   STATUS[3878] := 16#00;
   STATUS[3879] := 16#00;
   STATUS[3880] := 16#00;
   STATUS[3881] := 16#00;
   STATUS[3882] := 16#00;
   STATUS[3883] := 16#00;
   STATUS[3884] := 16#00;
   STATUS[3885] := 16#00;
   STATUS[3886] := 16#00;
   STATUS[3887] := 16#00;
   STATUS[3888] := 16#00;
   STATUS[3889] := 16#00;
   STATUS[3890] := 16#00;
   STATUS[3891] := 16#00;
   STATUS[3892] := 16#00;
   STATUS[3893] := 16#00;
   STATUS[3894] := 16#00;
   STATUS[3895] := 16#00;
   STATUS[3896] := 16#00;
   STATUS[3897] := 16#00;
   STATUS[3898] := 16#00;
   STATUS[3899] := 16#00;
   STATUS[3900] := 16#00;
   STATUS[3901] := 16#00;
   STATUS[3902] := 16#00;
   STATUS[3903] := 16#00;
   STATUS[3904] := 16#00;
   STATUS[3905] := 16#00;
   STATUS[3906] := 16#00;
   STATUS[3907] := 16#00;
   STATUS[3908] := 16#00;
   STATUS[3909] := 16#00;
   STATUS[3910] := 16#00;
   STATUS[3911] := 16#00;
   STATUS[3912] := 16#00;
   STATUS[3913] := 16#00;
   STATUS[3914] := 16#00;
   STATUS[3915] := 16#00;
   STATUS[3916] := 16#00;
   STATUS[3917] := 16#00;
   STATUS[3918] := 16#00;
   STATUS[3919] := 16#00;
   STATUS[3920] := 16#00;
   STATUS[3921] := 16#00;
   STATUS[3922] := 16#00;
   STATUS[3923] := 16#00;
   STATUS[3924] := 16#00;
   STATUS[3925] := 16#00;
   STATUS[3926] := 16#00;
   STATUS[3927] := 16#00;
   STATUS[3928] := 16#00;
   STATUS[3929] := 16#00;
   STATUS[3930] := 16#00;
   STATUS[3931] := 16#00;
   STATUS[3932] := 16#00;
   STATUS[3933] := 16#00;
   STATUS[3934] := 16#00;
   STATUS[3935] := 16#00;
   STATUS[3936] := 16#00;
   STATUS[3937] := 16#00;
   STATUS[3938] := 16#00;
   STATUS[3939] := 16#00;
   STATUS[3940] := 16#00;
   STATUS[3941] := 16#00;
   STATUS[3942] := 16#00;
   STATUS[3943] := 16#00;
   STATUS[3944] := 16#00;
   STATUS[3945] := 16#00;
   STATUS[3946] := 16#00;
   STATUS[3947] := 16#00;
   STATUS[3948] := 16#00;
   STATUS[3949] := 16#00;
   STATUS[3950] := 16#00;
   STATUS[3951] := 16#00;
   STATUS[3952] := 16#00;
   STATUS[3953] := 16#00;
   STATUS[3954] := 16#00;
   STATUS[3955] := 16#00;
   STATUS[3956] := 16#00;
   STATUS[3957] := 16#00;
   STATUS[3958] := 16#00;
   STATUS[3959] := 16#00;
   STATUS[3960] := 16#00;
   STATUS[3961] := 16#00;
   STATUS[3962] := 16#00;
   STATUS[3963] := 16#00;
   STATUS[3964] := 16#00;
   STATUS[3965] := 16#00;
   STATUS[3966] := 16#00;
   STATUS[3967] := 16#00;
   STATUS[3968] := 16#00;
   STATUS[3969] := 16#00;
   STATUS[3970] := 16#00;
   STATUS[3971] := 16#00;
   STATUS[3972] := 16#00;
   STATUS[3973] := 16#00;
   STATUS[3974] := 16#00;
   STATUS[3975] := 16#00;
   STATUS[3976] := 16#00;
   STATUS[3977] := 16#00;
   STATUS[3978] := 16#00;
   STATUS[3979] := 16#00;
   STATUS[3980] := 16#00;
   STATUS[3981] := 16#00;
   STATUS[3982] := 16#00;
   STATUS[3983] := 16#00;
   STATUS[3984] := 16#00;
   STATUS[3985] := 16#00;
   STATUS[3986] := 16#00;
   STATUS[3987] := 16#00;
   STATUS[3988] := 16#00;
   STATUS[3989] := 16#00;
   STATUS[3990] := 16#00;
   STATUS[3991] := 16#00;
   STATUS[3992] := 16#00;
   STATUS[3993] := 16#00;
   STATUS[3994] := 16#00;
   STATUS[3995] := 16#00;
   STATUS[3996] := 16#00;
   STATUS[3997] := 16#00;
   STATUS[3998] := 16#00;
   STATUS[3999] := 16#00;
   STATUS[4000] := 16#00;
   STATUS[4001] := 16#00;
   STATUS[4002] := 16#00;
   STATUS[4003] := 16#00;
   STATUS[4004] := 16#00;
   STATUS[4005] := 16#00;
   STATUS[4006] := 16#00;
   STATUS[4007] := 16#00;
   STATUS[4008] := 16#00;
   STATUS[4009] := 16#00;
   STATUS[4010] := 16#00;
   STATUS[4011] := 16#00;
   STATUS[4012] := 16#00;
   STATUS[4013] := 16#00;
   STATUS[4014] := 16#00;
   STATUS[4015] := 16#00;
   STATUS[4016] := 16#00;
   STATUS[4017] := 16#00;
   STATUS[4018] := 16#00;
   STATUS[4019] := 16#00;
   STATUS[4020] := 16#00;
   STATUS[4021] := 16#00;
   STATUS[4022] := 16#00;
   STATUS[4023] := 16#00;
   STATUS[4024] := 16#00;
   STATUS[4025] := 16#00;
   STATUS[4026] := 16#00;
   STATUS[4027] := 16#00;
   STATUS[4028] := 16#00;
   STATUS[4029] := 16#00;
   STATUS[4030] := 16#00;
   STATUS[4031] := 16#00;
   STATUS[4032] := 16#00;
   STATUS[4033] := 16#00;
   STATUS[4034] := 16#00;
   STATUS[4035] := 16#00;
   STATUS[4036] := 16#00;
   STATUS[4037] := 16#00;
   STATUS[4038] := 16#00;
   STATUS[4039] := 16#00;
   STATUS[4040] := 16#00;
   STATUS[4041] := 16#00;
   STATUS[4042] := 16#00;
   STATUS[4043] := 16#00;
   STATUS[4044] := 16#00;
   STATUS[4045] := 16#00;
   STATUS[4046] := 16#00;
   STATUS[4047] := 16#00;
   STATUS[4048] := 16#00;
   STATUS[4049] := 16#00;
   STATUS[4050] := 16#00;
   STATUS[4051] := 16#00;
   STATUS[4052] := 16#00;
   STATUS[4053] := 16#00;
   STATUS[4054] := 16#00;
   STATUS[4055] := 16#00;
   STATUS[4056] := 16#00;
   STATUS[4057] := 16#00;
   STATUS[4058] := 16#00;
   STATUS[4059] := 16#00;
   STATUS[4060] := 16#00;
   STATUS[4061] := 16#00;
   STATUS[4062] := 16#00;
   STATUS[4063] := 16#00;
   STATUS[4064] := 16#00;
   STATUS[4065] := 16#00;
   STATUS[4066] := 16#00;
   STATUS[4067] := 16#00;
   STATUS[4068] := 16#00;
   STATUS[4069] := 16#00;
   STATUS[4070] := 16#00;
   STATUS[4071] := 16#00;
   STATUS[4072] := 16#00;
   STATUS[4073] := 16#00;
   STATUS[4074] := 16#00;
   STATUS[4075] := 16#00;
   STATUS[4076] := 16#00;
   STATUS[4077] := 16#00;
   STATUS[4078] := 16#00;
   STATUS[4079] := 16#00;
   STATUS[4080] := 16#00;
   STATUS[4081] := 16#00;
   STATUS[4082] := 16#00;
   STATUS[4083] := 16#00;
   STATUS[4084] := 16#00;
   STATUS[4085] := 16#00;
   STATUS[4086] := 16#00;
   STATUS[4087] := 16#00;
   STATUS[4088] := 16#00;
   STATUS[4089] := 16#00;
   STATUS[4090] := 16#00;
   STATUS[4091] := 16#00;
   STATUS[4092] := 16#00;
   STATUS[4093] := 16#00;
   STATUS[4094] := 16#00;
   STATUS[4095] := 16#00;
   STATUS[4096] := 16#00;
END_DATA_BLOCK

DATA_BLOCK "ACESYS_HMI_INDICATION"   // DB11
TITLE = Boolean Indications to HMI
{ S7_Optimized_Access := 'FALSE' }
AUTHOR : METIS
FAMILY : ACESYS
NAME : IndDB
VERSION : 8.0
   VAR
      "997CD100D01_RESET_ALRM" : Bool := FALSE;   // Reset Alarm In Area
      "2010BF110U01_STOP_FROM_ECS" : Bool := FALSE;   // Ext Stop From ECS
      "2010HP100TL01CMD01" : Bool := FALSE;   // Переключение сигнала сфетофора
      "2010HP100TL01GRN01" : Bool := FALSE;   // Светофор красный
      "2010HP100TL01RED01" : Bool := TRUE;   // Светофор красный
      "2010BF110U01_SPD_UP" : Bool := FALSE;   // Увеличить задание на 1
      "2010BF110U01_SPD_DN" : Bool := TRUE;   // Уменьшить задание на 1
      "3015PU040_042_OFF" : Bool := FALSE;
      "2010HP100TL01CMD2" : Bool := FALSE;   // Светофор Включить зелёный
      "2010HP100TL01CMD3" : Bool := FALSE;   // Светофор Включить красный
      IND11 : Bool := FALSE;
      IND12 : Bool := TRUE;
      IND13 : Bool := FALSE;
      IND14 : Bool := FALSE;
      IND15 : Bool := FALSE;
      IND16 : Bool := TRUE;
      IND17 : Bool := FALSE;
      IND18 : Bool := FALSE;
      IND19 : Bool := FALSE;
      "2010SJ950M01_ASTR" : Bool := FALSE;
      IND21 : Bool := FALSE;
      IND22 : Bool := FALSE;
      IND23 : Bool := FALSE;
      IND24 : Bool := FALSE;
      IND25 : Bool := FALSE;
      IND26 : Bool := FALSE;
      IND27 : Bool := FALSE;
      IND28 : Bool := TRUE;
      IND29 : Bool := FALSE;
      IND30 : Bool := FALSE;
      IND31 : Bool := FALSE;
      IND32 : Bool := FALSE;
      IND33 : Bool := FALSE;
      IND34 : Bool := FALSE;
      IND35 : Bool := FALSE;
      IND36 : Bool := FALSE;
      IND37 : Bool := FALSE;
      IND38 : Bool := FALSE;
      IND39 : Bool := FALSE;
      IND40 : Bool := FALSE;
      IND41 : Bool := FALSE;
      IND42 : Bool := FALSE;
      IND43 : Bool := TRUE;
      IND44 : Bool := TRUE;
      IND45 : Bool := FALSE;
      IND46 : Bool := FALSE;
      IND47 : Bool := FALSE;
      IND48 : Bool := FALSE;
      IND49 : Bool := FALSE;
      IND50 : Bool := FALSE;
      IND51 : Bool := FALSE;
      IND52 : Bool := FALSE;
      IND53 : Bool := FALSE;
      IND54 : Bool := TRUE;
      IND55 : Bool := FALSE;
      IND56 : Bool := TRUE;
      IND57 : Bool := TRUE;
      IND58 : Bool := TRUE;
      IND59 : Bool := FALSE;
      _995CS100_INDICATION01 : Bool := FALSE;   // INDICATION01
      _995CS100_INDICATION02 : Bool := FALSE;   // INDICATION02
      _995CS100_INDICATION03 : Bool := FALSE;   // INDICATION03
      _995CS100_INDICATION04 : Bool := FALSE;   // INDICATION04
      _995CS100_INDICATION05 : Bool := FALSE;   // INDICATION05
      _995CS100_INDICATION06 : Bool := FALSE;   // INDICATION06
      _995CS100_INDICATION07 : Bool := FALSE;   // INDICATION07
      _995CS100_INDICATION08 : Bool := FALSE;   // INDICATION08
      _995CS100_INDICATION09 : Bool := FALSE;   // INDICATION09
      _995CS100_INDICATION10 : Bool := FALSE;   // INDICATION10
      _995CS100_INDICATION11 : Bool := FALSE;   // INDICATION11
      _995CS100_INDICATION12 : Bool := FALSE;   // INDICATION12
      _995CS100_INDICATION13 : Bool := FALSE;   // INDICATION13
      _995CS100_INDICATION14 : Bool := FALSE;   // INDICATION14
      _995CS100_INDICATION15 : Bool := FALSE;   // INDICATION15
      _995CS100_INDICATION16 : Bool := FALSE;   // INDICATION16
      _995CS100_INDICATION17 : Bool := FALSE;   // INDICATION17
      _995CS100_INDICATION18 : Bool := FALSE;   // INDICATION18
      _995CS100_INDICATION19 : Bool := FALSE;   // INDICATION19
      _995CS100_INDICATION20 : Bool := FALSE;   // INDICATION20
      _995CS100_INDICATION21 : Bool := FALSE;   // INDICATION21
      _995CS100_INDICATION22 : Bool := FALSE;   // INDICATION22
      _995CS100_INDICATION23 : Bool := FALSE;   // INDICATION23
      _995CS100_INDICATION24 : Bool := FALSE;   // INDICATION24
      _995CS100_INDICATION25 : Bool := FALSE;   // INDICATION25
      _995CS100_INDICATION26 : Bool := FALSE;   // INDICATION26
      _995CS100_INDICATION27 : Bool := FALSE;   // INDICATION27
      _995CS100_INDICATION28 : Bool := FALSE;   // INDICATION28
      _995CS100_INDICATION29 : Bool := FALSE;   // INDICATION29
      _995CS100_INDICATION30 : Bool := FALSE;   // INDICATION30
      _995CS100_INDICATION31 : Bool := FALSE;   // INDICATION31
      _995CS100_INDICATION32 : Bool := FALSE;   // INDICATION32
      _995CS100_INDICATION33 : Bool := FALSE;   // INDICATION33
      _995CS100_INDICATION34 : Bool := FALSE;   // INDICATION34
      _995CS100_INDICATION35 : Bool := FALSE;   // INDICATION35
      _995CS100_INDICATION36 : Bool := FALSE;   // INDICATION36
      _995CS100_INDICATION37 : Bool := FALSE;   // INDICATION37
      _995CS100_INDICATION38 : Bool := FALSE;   // INDICATION38
      _995CS100_INDICATION39 : Bool := FALSE;   // INDICATION39
      _995CS100_INDICATION40 : Bool := FALSE;   // INDICATION40
      _995CS100_INDICATION41 : Bool := FALSE;   // INDICATION41
      _995CS100_INDICATION42 : Bool := FALSE;   // INDICATION42
      _995CS100_INDICATION43 : Bool := FALSE;   // INDICATION43
      _995CS100_INDICATION44 : Bool := FALSE;   // INDICATION44
      _995CS100_INDICATION45 : Bool := FALSE;   // INDICATION45
      _995CS100_INDICATION46 : Bool := FALSE;   // INDICATION46
      _995CS100_INDICATION47 : Bool := FALSE;   // INDICATION47
      _995CS100_INDICATION48 : Bool := FALSE;   // INDICATION48
      _995CS100_INDICATION49 : Bool := FALSE;   // INDICATION49
      _995CS100_INDICATION50 : Bool := FALSE;   // INDICATION50
      _995CS100_SIMPLEINDI01 : Bool := FALSE;   // SIMPLEINDI01
      _995CS100_SIMPLEINDI02 : Bool := FALSE;   // SIMPLEINDI02
      _995CS100_SIMPLEINDI03 : Bool := FALSE;   // SIMPLEINDI03
      _995CS100_SIMPLEINDI04 : Bool := FALSE;   // SIMPLEINDI04
      _995CS100_SIMPLEINDI05 : Bool := FALSE;   // SIMPLEINDI05
      _995CS100_SIMPLEINDI06 : Bool := FALSE;   // SIMPLEINDI06
      _995CS100_SIMPLEINDI07 : Bool := FALSE;   // SIMPLEINDI07
      _995CS100_SIMPLEINDI08 : Bool := FALSE;   // SIMPLEINDI08
      _995CS100_SIMPLEINDI09 : Bool := FALSE;   // SIMPLEINDI09
      _995CS100_SIMPLEINDI10 : Bool := FALSE;   // SIMPLEINDI10
      _995CS100_SIMPLEINDI11 : Bool := FALSE;   // SIMPLEINDI11
      _995CS100_SIMPLEINDI12 : Bool := FALSE;   // SIMPLEINDI12
      _995CS100_SIMPLEINDI13 : Bool := FALSE;   // SIMPLEINDI13
      _995CS100_SIMPLEINDI14 : Bool := FALSE;   // SIMPLEINDI14
      _995CS100_SIMPLEINDI15 : Bool := FALSE;   // SIMPLEINDI15
      _995CS100_SIMPLEINDI16 : Bool := FALSE;   // SIMPLEINDI16
      _995CS100_SIMPLEINDI17 : Bool := FALSE;   // SIMPLEINDI17
      _995CS100_SIMPLEINDI18 : Bool := FALSE;   // SIMPLEINDI18
      _995CS100_SIMPLEINDI19 : Bool := FALSE;   // SIMPLEINDI19
      _995CS100_SIMPLEINDI20 : Bool := FALSE;   // SIMPLEINDI20
   END_VAR
BEGIN
END_DATA_BLOCK

DATA_BLOCK "ACESYS_HMI_OPERATORSP"   // DB12
TITLE = Simple setpoints from HMI
{ S7_Optimized_Access := 'FALSE' }
AUTHOR : METIS
FAMILY : ACESYS
NAME : OpDB
VERSION : 8.0
   VAR
      _2010CV300U01_SP : Real := 120.0;   // Set Spd CV300
      _2010CV180U01_SP : Real := 100.0;   // Set Speed
      _spare : Real := 0.0;   // Set Speed
      _2010BF110U01_SP : Real := 0.0;   // Set Speed
      _2010SC130U01_SP : Real := 100.0;   // Set Speed
      _MTR_SPARE_SP : Real := 110.0;
      spare_6 : Real := 70.0;
      spare_7 : Real := 0.0;
      spare_8 : Real := 0.0;
      spare_9 : Real := 0.0;
      spare_10 : Real := 0.0;
      spare_11 : Real := 0.0;
      spare_12 : Real := 0.0;
      spare_13 : Real := 0.0;
      spare_14 : Real := 0.0;   // OPERATORSP01
      spare_15 : Real := 0.0;   // OPERATORSP02
      spare_16 : Real := 0.0;   // OPERATORSP03
      spare_17 : Real := 0.0;   // OPERATORSP04
      spare_18 : Real := 0.0;   // OPERATORSP05
      spare_19 : Real := 0.0;   // OPERATORSP06
      spare_20 : Real := 0.0;   // OPERATORSP07
      spare_21 : Real := 0.0;   // OPERATORSP08
      spare_22 : Real := 0.0;   // OPERATORSP09
      spare_23 : Real := 0.0;   // OPERATORSP10
      spare_24 : Real := 0.0;   // OPERATORSP11
      spare_25 : Real := 0.0;   // OPERATORSP12
      spare_26 : Real := 0.0;   // OPERATORSP13
      spare_27 : Real := 0.0;   // OPERATORSP14
      spare_28 : Real := 0.0;   // OPERATORSP15
      spare_29 : Real := 0.0;   // OPERATORSP16
      spare_30 : Real := 0.0;   // OPERATORSP17
      spare_31 : Real := 0.0;   // OPERATORSP18
      spare_32 : Real := 0.0;   // OPERATORSP19
      spare_33 : Real := 0.0;   // OPERATORSP20
      spare_34 : Real := 0.0;   // OPERATORSP21
      spare_35 : Real := 0.0;   // OPERATORSP22
      spare_36 : Real := 0.0;   // OPERATORSP23
      spare_37 : Real := 0.0;   // OPERATORSP24
      spare_38 : Real := 0.0;   // OPERATORSP25
      spare_39 : Real := 0.0;   // OPERATORSP26
      spare_40 : Real := 0.0;   // OPERATORSP27
      spare_41 : Real := 0.0;   // OPERATORSP28
      spare_42 : Real := 0.0;   // OPERATORSP29
      spare_43 : Real := 0.0;   // OPERATORSP30
   END_VAR
BEGIN
END_DATA_BLOCK

DATA_BLOCK "ACESYS_HMI_SIMPLEAI"   // DB13
TITLE = Simple Analog Values to HMI
{ S7_Optimized_Access := 'FALSE' }
AUTHOR : METIS
FAMILY : ACESYS
NAME : AiDB
VERSION : 8.0
   VAR
      _997CS100_Sec : Real := 16#0000_001A;   // CPU Clock Seconds
      _997CS100_Min : Real := 16#0000_0009;   // CPU Clock Minutes
      _997CS100_Hour : Real := 16#0000_000E;   // CPU Clock Hours
      _997CS100_Day : Real := 16#0000_0009;   // CPU Clock Day
      _997CS100_Month : Real := 16#0000_0003;   // CPU Clock Month
      _997CS100_Year : Real := 16#0000_0019;   // CPU Clock Year
      _997CS100_MemTot : Real := 1.884792E-29;   // Total CPU Memory
      _997CS100_MemUsed : Real := 1.715889E-38;   // Used CPU Memory
      _997CS100_MemPct : Real := 4.63501;   // Used CPU Memory
      _2015PU040U01_AO1b : Real := 10.64;
      _2015PU040U01_AO3a : Real := 80.005;
      _2015PU041U01_AO1b : Real := 0.0;
      _2015PU041U01_AO3a : Real := 0.0;
      _2015PU042U01_AO1b : Real := 4.361;
      _2015PU027U01_AO1b : Real := 0.0;
      _2015PU027U01_AO3a : Real := 0.0;
      _2015PU028U01_AO1b : Real := 0.0;
      _2015PU028U01_AO3a : Real := 0.0;
      _2015PU035U01_AO1b : Real := 0.0;
      _2015PU035U01_AO3a : Real := 0.0;
      _2010SJ950M01_AO1b : Real := 0.0;
      _993CS100_ANALOGINDI22 : Real := 700.0326;
      _993CS100_ANALOGINDI23 : Real := 0.0;
      _993CS100_ANALOGINDI24 : Real := 0.0;
      _993CS100_ANALOGINDI25 : Real := 0.0;
      _993CS100_ANALOGINDI26 : Real := 0.0;
      _993CS100_ANALOGINDI27 : Real := 0.0;
      _993CS100_ANALOGINDI28 : Real := 0.0;
      _993CS100_ANALOGINDI29 : Real := 0.0;
      _993CS100_ANALOGINDI30 : Real := 0.0;
      _993CS100_ANALOGINDI31 : Real := 0.0;
      _993CS100_ANALOGINDI32 : Real := 0.0;
      _993CS100_ANALOGINDI33 : Real := 0.0;
      _993CS100_ANALOGINDI34 : Real := 0.0;
      _993CS100_ANALOGINDI35 : Real := 0.0;
      _993CS100_ANALOGINDI36 : Real := 0.0;
      _993CS100_ANALOGINDI37 : Real := 0.0;
      _993CS100_ANALOGINDI38 : Real := 0.0;
      _993CS100_ANALOGINDI39 : Real := 0.0;
      _993CS100_ANALOGINDI40 : Real := 0.0;
      _993CS100_ANALOGINDI41 : Real := 0.0;
      _993CS100_ANALOGINDI42 : Real := 0.0;
      _993CS100_ANALOGINDI43 : Real := 0.0;
      _993CS100_ANALOGINDI44 : Real := 0.0;
      _993CS100_ANALOGINDI45 : Real := 0.0;
      _993CS100_ANALOGINDI46 : Real := 0.0;
      _993CS100_ANALOGINDI47 : Real := 0.0;
      _993CS100_ANALOGINDI48 : Real := 0.0;
      _993CS100_ANALOGINDI49 : Real := 0.0;
      _993CS100_ANALOGINDI50 : Real := 16#0000_003C;   // OB1 Scan Time
      _993CS100_ANALOGINDI51 : Real := 16#0000_0064;   // OB35 Scan Time
      _993CS100_ANALOGINDI52 : Real := 0.0;
      _993CS100_ANALOGINDI53 : Real := 0.0;
      _993CS100_ANALOGINDI54 : Real := 0.0;
      _993CS100_ANALOGINDI55 : Real := 0.0;
      _993CS100_ANALOGINDI56 : Real := 0.0;
      _993CS100_ANALOGINDI57 : Real := 0.0;
      _993CS100_ANALOGINDI58 : Real := 0.0;
      _993CS100_ANALOGINDI59 : Real := 0.0;
      _2010LV100P01_I1 : Real := 7.9433;
      _2010LV100P01_I2 : Real := 9.236307;
      _2010LV100P01_I3 : Real := 6.303556;
      _2010LV100P01_E01 : Real := 412.6258;
      _2010LV100P01_E02 : Real := 411.3553;
      _2010LV100P01_E03 : Real := 412.2155;
      _2010LV100P01_X01 : Real := 49.99622;
      _2010LV100P01_X02 : Real := 0.8079877;
      _2010LV100P01_J1 : Real := 5.585882;
      _2010LV100P01_J2 : Real := 4.513324;
      _2010LV100P01_J3 : Real := 2.662353;
      _2010LV100P01_Q01 : Real := 1852637.0;
      _2010LV100P01_Q02 : Real := 355350.2;
      _2010LV100P01_Q03 : Real := 2301733.0;
      _993CS100_ANALOGINDI74 : Real := 0.0;
      _993CS100_ANALOGINDI75 : Real := 0.0;
      _993CS100_ANALOGINDI76 : Real := 0.0;
      _993CS100_ANALOGINDI77 : Real := 0.0;
      _993CS100_ANALOGINDI78 : Real := 0.0;
      _993CS100_ANALOGINDI79 : Real := 0.0;
      _993CS100_ANALOGINDI80 : Real := 0.0;
      _993CS100_ANALOGINDI81 : Real := 0.0;
   END_VAR
BEGIN
END_DATA_BLOCK

DATA_BLOCK "ACESYS_HMI_SIMPLEREQ"   // DB14
TITLE = Simple Binary Requests from HMI
{ S7_Optimized_Access := 'FALSE' }
AUTHOR : METIS
FAMILY : ACESYS
NAME : BinReq
VERSION : 8.0
   VAR
      _995CS100HLC_CCA1 : Bool := FALSE;   // Computer Control Accept (Group 1-5)
      _995CS100HLC_CCA1_1 : Bool := FALSE;   // Dont use Bit 1
      _995CS100HLC_CCA1_2 : Bool := FALSE;   // Dont use Bit 2
      _995CS100HLC_CCA1_3 : Bool := FALSE;   // Dont use Bit 3
      _995CS100HLC_CCA1_4 : Bool := FALSE;   // Dont use Bit 4
      _995CS100HLC_CCA1_5 : Bool := FALSE;   // Dont use Bit 5
      _995CS100HLC_CCA1_6 : Bool := FALSE;   // Dont use Bit 6
      _995CS100HLC_CCA1_7 : Bool := FALSE;   // Dont use Bit 7
      _995CS100HLC_CCA2 : Bool := FALSE;   // Computer Control Accept (Group 6-10)
      _995CS100HLC_CCA2_1 : Bool := FALSE;   // Dont use Bit 1
      _995CS100HLC_CCA2_2 : Bool := FALSE;   // Dont use Bit 2
      _995CS100HLC_CCA2_3 : Bool := FALSE;   // Dont use Bit 3
      _995CS100HLC_CCA2_4 : Bool := FALSE;   // Dont use Bit 4
      _995CS100HLC_CCA2_5 : Bool := FALSE;   // Dont use Bit 5
      _995CS100HLC_CCA2_6 : Bool := FALSE;   // Dont use Bit 6
      _995CS100HLC_CCA2_7 : Bool := FALSE;   // Dont use Bit 7
      _995CS100HLC_KA : Bool := FALSE;   // Keep Alive (Watchdog)
      _995CS100HLC_KA_1 : Bool := FALSE;   // Dont use Bit 1
      _995CS100HLC_KA_2 : Bool := FALSE;   // Dont use Bit 2
      _995CS100HLC_KA_3 : Bool := FALSE;   // Dont use Bit 3
      _995CS100HLC_KA_4 : Bool := FALSE;   // Dont use Bit 4
      _995CS100HLC_KA_5 : Bool := FALSE;   // Dont use Bit 5
      _995CS100HLC_KA_6 : Bool := FALSE;   // Dont use Bit 6
      _995CS100HLC_KA_7 : Bool := FALSE;   // Dont use Bit 7
      _995CS100HLC_GRP01 : Bool := FALSE;   // HLC Group 01 Enabled
      _995CS100HLC_GRP01_1 : Bool := FALSE;   // Dont use Bit 7
      _995CS100HLC_GRP01_2 : Bool := FALSE;   // Dont use Bit 2
      _995CS100HLC_GRP01_3 : Bool := FALSE;   // Dont use Bit 3
      _995CS100HLC_GRP01_4 : Bool := FALSE;   // Dont use Bit 4
      _995CS100HLC_GRP01_5 : Bool := FALSE;   // Dont use Bit 5
      _995CS100HLC_GRP01_6 : Bool := FALSE;   // Dont use Bit 6
      _995CS100HLC_GRP01_7 : Bool := FALSE;   // Dont use Bit 7
      _995CS100HLC_GRP02 : Bool := FALSE;   // HLC Group 02 Enabled
      _995CS100HLC_GRP02_1 : Bool := FALSE;   // Dont use Bit 7
      _995CS100HLC_GRP02_2 : Bool := FALSE;   // Dont use Bit 2
      _995CS100HLC_GRP02_3 : Bool := FALSE;   // Dont use Bit 3
      _995CS100HLC_GRP02_4 : Bool := FALSE;   // Dont use Bit 4
      _995CS100HLC_GRP02_5 : Bool := FALSE;   // Dont use Bit 5
      _995CS100HLC_GRP02_6 : Bool := FALSE;   // Dont use Bit 6
      _995CS100HLC_GRP02_7 : Bool := FALSE;   // Dont use Bit 7
      _995CS100HLC_GRP03 : Bool := FALSE;   // HLC Group 03 Enabled
      _995CS100HLC_GRP03_1 : Bool := FALSE;   // Dont use Bit 7
      _995CS100HLC_GRP03_2 : Bool := FALSE;   // Dont use Bit 2
      _995CS100HLC_GRP03_3 : Bool := FALSE;   // Dont use Bit 3
      _995CS100HLC_GRP03_4 : Bool := FALSE;   // Dont use Bit 4
      _995CS100HLC_GRP03_5 : Bool := FALSE;   // Dont use Bit 5
      _995CS100HLC_GRP03_6 : Bool := FALSE;   // Dont use Bit 6
      _995CS100HLC_GRP03_7 : Bool := FALSE;   // Dont use Bit 7
      _995CS100HLC_GRP04 : Bool := FALSE;   // HLC Group 04 Enabled
      _995CS100HLC_GRP04_1 : Bool := FALSE;   // Dont use Bit 7
      _995CS100HLC_GRP04_2 : Bool := FALSE;   // Dont use Bit 2
      _995CS100HLC_GRP04_3 : Bool := FALSE;   // Dont use Bit 3
      _995CS100HLC_GRP04_4 : Bool := FALSE;   // Dont use Bit 4
      _995CS100HLC_GRP04_5 : Bool := FALSE;   // Dont use Bit 5
      _995CS100HLC_GRP04_6 : Bool := FALSE;   // Dont use Bit 6
      _995CS100HLC_GRP04_7 : Bool := FALSE;   // Dont use Bit 7
      _995CS100HLC_GRP05 : Bool := FALSE;   // HLC Group 05 Enabled
      _995CS100HLC_GRP05_1 : Bool := FALSE;   // Dont use Bit 7
      _995CS100HLC_GRP05_2 : Bool := FALSE;   // Dont use Bit 2
      _995CS100HLC_GRP05_3 : Bool := FALSE;   // Dont use Bit 3
      _995CS100HLC_GRP05_4 : Bool := FALSE;   // Dont use Bit 4
      _995CS100HLC_GRP05_5 : Bool := FALSE;   // Dont use Bit 5
      _995CS100HLC_GRP05_6 : Bool := FALSE;   // Dont use Bit 6
      _995CS100HLC_GRP05_7 : Bool := FALSE;   // Dont use Bit 7
      _995CS100HLC_GRP06 : Bool := FALSE;   // HLC Group 06 Enabled
      _995CS100HLC_GRP06_1 : Bool := FALSE;   // Dont use Bit 7
      _995CS100HLC_GRP06_2 : Bool := FALSE;   // Dont use Bit 2
      _995CS100HLC_GRP06_3 : Bool := FALSE;   // Dont use Bit 3
      _995CS100HLC_GRP06_4 : Bool := FALSE;   // Dont use Bit 4
      _995CS100HLC_GRP06_5 : Bool := FALSE;   // Dont use Bit 5
      _995CS100HLC_GRP06_6 : Bool := FALSE;   // Dont use Bit 6
      _995CS100HLC_GRP06_7 : Bool := FALSE;   // Dont use Bit 7
      _995CS100HLC_GRP07 : Bool := FALSE;   // HLC Group 07 Enabled
      _995CS100HLC_GRP07_1 : Bool := FALSE;   // Dont use Bit 7
      _995CS100HLC_GRP07_2 : Bool := FALSE;   // Dont use Bit 2
      _995CS100HLC_GRP07_3 : Bool := FALSE;   // Dont use Bit 3
      _995CS100HLC_GRP07_4 : Bool := FALSE;   // Dont use Bit 4
      _995CS100HLC_GRP07_5 : Bool := FALSE;   // Dont use Bit 5
      _995CS100HLC_GRP07_6 : Bool := FALSE;   // Dont use Bit 6
      _995CS100HLC_GRP07_7 : Bool := FALSE;   // Dont use Bit 7
      _995CS100HLC_GRP08 : Bool := FALSE;   // HLC Group 08 Enabled
      _995CS100HLC_GRP08_1 : Bool := FALSE;   // Dont use Bit 7
      _995CS100HLC_GRP08_2 : Bool := FALSE;   // Dont use Bit 2
      _995CS100HLC_GRP08_3 : Bool := FALSE;   // Dont use Bit 3
      _995CS100HLC_GRP08_4 : Bool := FALSE;   // Dont use Bit 4
      _995CS100HLC_GRP08_5 : Bool := FALSE;   // Dont use Bit 5
      _995CS100HLC_GRP08_6 : Bool := FALSE;   // Dont use Bit 6
      _995CS100HLC_GRP08_7 : Bool := FALSE;   // Dont use Bit 7
      _995CS100HLC_GRP09 : Bool := FALSE;   // HLC Group 09 Enabled
      _995CS100HLC_GRP09_1 : Bool := FALSE;   // Dont use Bit 7
      _995CS100HLC_GRP09_2 : Bool := FALSE;   // Dont use Bit 2
      _995CS100HLC_GRP09_3 : Bool := FALSE;   // Dont use Bit 3
      _995CS100HLC_GRP09_4 : Bool := FALSE;   // Dont use Bit 4
      _995CS100HLC_GRP09_5 : Bool := FALSE;   // Dont use Bit 5
      _995CS100HLC_GRP09_6 : Bool := FALSE;   // Dont use Bit 6
      _995CS100HLC_GRP09_7 : Bool := FALSE;   // Dont use Bit 7
      _995CS100HLC_GRP10 : Bool := FALSE;   // HLC Group 10 Enabled
      _995CS100HLC_GRP10_1 : Bool := FALSE;   // Dont use Bit 7
      _995CS100HLC_GRP10_2 : Bool := FALSE;   // Dont use Bit 2
      _995CS100HLC_GRP10_3 : Bool := FALSE;   // Dont use Bit 3
      _995CS100HLC_GRP10_4 : Bool := FALSE;   // Dont use Bit 4
      _995CS100HLC_GRP10_5 : Bool := FALSE;   // Dont use Bit 5
      _995CS100HLC_GRP10_6 : Bool := FALSE;   // Dont use Bit 6
      _995CS100HLC_GRP10_7 : Bool := FALSE;   // Dont use Bit 7
      _995CS100HLC_RDY01 : Bool := FALSE;   // HLC Group 01 Ready
      _995CS100HLC_RDY01_1 : Bool := FALSE;   // Dont use Bit 1
      _995CS100HLC_RDY01_2 : Bool := FALSE;   // Dont use Bit 2
      _995CS100HLC_RDY01_3 : Bool := FALSE;   // Dont use Bit 3
      _995CS100HLC_RDY01_4 : Bool := FALSE;   // Dont use Bit 4
      _995CS100HLC_RDY01_5 : Bool := FALSE;   // Dont use Bit 5
      _995CS100HLC_RDY01_6 : Bool := FALSE;   // Dont use Bit 6
      _995CS100HLC_RDY01_7 : Bool := FALSE;   // Dont use Bit 7
      _995CS100HLC_RDY02 : Bool := FALSE;   // HLC Group 02 Ready
      _995CS100HLC_RDY02_1 : Bool := FALSE;   // Dont use Bit 1
      _995CS100HLC_RDY02_2 : Bool := FALSE;   // Dont use Bit 2
      _995CS100HLC_RDY02_3 : Bool := FALSE;   // Dont use Bit 3
      _995CS100HLC_RDY02_4 : Bool := FALSE;   // Dont use Bit 4
      _995CS100HLC_RDY02_5 : Bool := FALSE;   // Dont use Bit 5
      _995CS100HLC_RDY02_6 : Bool := FALSE;   // Dont use Bit 6
      _995CS100HLC_RDY02_7 : Bool := FALSE;   // Dont use Bit 7
      _995CS100HLC_RDY03 : Bool := FALSE;   // HLC Group 03 Ready
      _995CS100HLC_RDY03_1 : Bool := FALSE;   // Dont use Bit 1
      _995CS100HLC_RDY03_2 : Bool := FALSE;   // Dont use Bit 2
      _995CS100HLC_RDY03_3 : Bool := FALSE;   // Dont use Bit 3
      _995CS100HLC_RDY03_4 : Bool := FALSE;   // Dont use Bit 4
      _995CS100HLC_RDY03_5 : Bool := FALSE;   // Dont use Bit 5
      _995CS100HLC_RDY03_6 : Bool := FALSE;   // Dont use Bit 6
      _995CS100HLC_RDY03_7 : Bool := FALSE;   // Dont use Bit 7
      _995CS100HLC_RDY04 : Bool := FALSE;   // HLC Group 04 Ready
      _995CS100HLC_RDY04_1 : Bool := FALSE;   // Dont use Bit 1
      _995CS100HLC_RDY04_2 : Bool := FALSE;   // Dont use Bit 2
      _995CS100HLC_RDY04_3 : Bool := FALSE;   // Dont use Bit 3
      _995CS100HLC_RDY04_4 : Bool := FALSE;   // Dont use Bit 4
      _995CS100HLC_RDY04_5 : Bool := FALSE;   // Dont use Bit 5
      _995CS100HLC_RDY04_6 : Bool := FALSE;   // Dont use Bit 6
      _995CS100HLC_RDY04_7 : Bool := FALSE;   // Dont use Bit 7
      _995CS100HLC_RDY05 : Bool := FALSE;   // HLC Group 05 Ready
      _995CS100HLC_RDY05_1 : Bool := FALSE;   // Dont use Bit 1
      _995CS100HLC_RDY05_2 : Bool := FALSE;   // Dont use Bit 2
      _995CS100HLC_RDY05_3 : Bool := FALSE;   // Dont use Bit 3
      _995CS100HLC_RDY05_4 : Bool := FALSE;   // Dont use Bit 4
      _995CS100HLC_RDY05_5 : Bool := FALSE;   // Dont use Bit 5
      _995CS100HLC_RDY05_6 : Bool := FALSE;   // Dont use Bit 6
      _995CS100HLC_RDY05_7 : Bool := FALSE;   // Dont use Bit 7
      _995CS100HLC_RDY06 : Bool := FALSE;   // HLC Group 06 Ready
      _995CS100HLC_RDY06_1 : Bool := FALSE;   // Dont use Bit 1
      _995CS100HLC_RDY06_2 : Bool := FALSE;   // Dont use Bit 2
      _995CS100HLC_RDY06_3 : Bool := FALSE;   // Dont use Bit 3
      _995CS100HLC_RDY06_4 : Bool := FALSE;   // Dont use Bit 4
      _995CS100HLC_RDY06_5 : Bool := FALSE;   // Dont use Bit 5
      _995CS100HLC_RDY06_6 : Bool := FALSE;   // Dont use Bit 6
      _995CS100HLC_RDY06_7 : Bool := FALSE;   // Dont use Bit 7
      _995CS100HLC_RDY07 : Bool := FALSE;   // HLC Group 07 Ready
      _995CS100HLC_RDY07_1 : Bool := FALSE;   // Dont use Bit 1
      _995CS100HLC_RDY07_2 : Bool := FALSE;   // Dont use Bit 2
      _995CS100HLC_RDY07_3 : Bool := FALSE;   // Dont use Bit 3
      _995CS100HLC_RDY07_4 : Bool := FALSE;   // Dont use Bit 4
      _995CS100HLC_RDY07_5 : Bool := FALSE;   // Dont use Bit 5
      _995CS100HLC_RDY07_6 : Bool := FALSE;   // Dont use Bit 6
      _995CS100HLC_RDY07_7 : Bool := FALSE;   // Dont use Bit 7
      _995CS100HLC_RDY08 : Bool := FALSE;   // HLC Group 08 Ready
      _995CS100HLC_RDY08_1 : Bool := FALSE;   // Dont use Bit 1
      _995CS100HLC_RDY08_2 : Bool := FALSE;   // Dont use Bit 2
      _995CS100HLC_RDY08_3 : Bool := FALSE;   // Dont use Bit 3
      _995CS100HLC_RDY08_4 : Bool := FALSE;   // Dont use Bit 4
      _995CS100HLC_RDY08_5 : Bool := FALSE;   // Dont use Bit 5
      _995CS100HLC_RDY08_6 : Bool := FALSE;   // Dont use Bit 6
      _995CS100HLC_RDY08_7 : Bool := FALSE;   // Dont use Bit 7
      _995CS100HLC_RDY09 : Bool := FALSE;   // HLC Group 09 Ready
      _995CS100HLC_RDY09_1 : Bool := FALSE;   // Dont use Bit 1
      _995CS100HLC_RDY09_2 : Bool := FALSE;   // Dont use Bit 2
      _995CS100HLC_RDY09_3 : Bool := FALSE;   // Dont use Bit 3
      _995CS100HLC_RDY09_4 : Bool := FALSE;   // Dont use Bit 4
      _995CS100HLC_RDY09_5 : Bool := FALSE;   // Dont use Bit 5
      _995CS100HLC_RDY09_6 : Bool := FALSE;   // Dont use Bit 6
      _995CS100HLC_RDY09_7 : Bool := FALSE;   // Dont use Bit 7
      _995CS100HLC_RDY10 : Bool := FALSE;   // HLC Group 10 Ready
      _995CS100HLC_RDY10_1 : Bool := FALSE;   // Dont use Bit 1
      _995CS100HLC_RDY10_2 : Bool := FALSE;   // Dont use Bit 2
      _995CS100HLC_RDY10_3 : Bool := FALSE;   // Dont use Bit 3
      _995CS100HLC_RDY10_4 : Bool := FALSE;   // Dont use Bit 4
      _995CS100HLC_RDY10_5 : Bool := FALSE;   // Dont use Bit 5
      _995CS100HLC_RDY10_6 : Bool := FALSE;   // Dont use Bit 6
      _995CS100HLC_RDY10_7 : Bool := FALSE;   // Dont use Bit 7
      _2090KL645A01REQ01 : Bool := FALSE;   // Reset System Alarm
      _2090KL645A01REQ011 : Bool := FALSE;   // Dont use Bit 1
      _2090KL645A01REQ012 : Bool := FALSE;   // Dont use Bit 2
      _2090KL645A01REQ013 : Bool := FALSE;   // Dont use Bit 3
      _2090KL645A01REQ014 : Bool := FALSE;   // Dont use Bit 4
      _2090KL645A01REQ015 : Bool := FALSE;   // Dont use Bit 5
      _2090KL645A01REQ016 : Bool := FALSE;   // Dont use Bit 6
      _2090KL645A01REQ017 : Bool := FALSE;   // Dont use Bit 7
      _3015SU026I01AUTH : Bool := FALSE;   // CS Feed Pump 1 Flow Control
      _3015SU026I01AUTH1 : Bool := FALSE;   // Dont use Bit 1
      _3015SU026I01AUTH2 : Bool := FALSE;   // Dont use Bit 2
      _3015SU026I01AUTH3 : Bool := FALSE;   // Dont use Bit 3
      _3015SU026I01AUTH4 : Bool := FALSE;   // Dont use Bit 4
      _3015SU026I01AUTH5 : Bool := FALSE;   // Dont use Bit 5
      _3015SU026I01AUTH6 : Bool := FALSE;   // Dont use Bit 6
      _3015SU026I01AUTH7 : Bool := FALSE;   // Dont use Bit 7
      _2090PU736I01AUTH : Bool := FALSE;   // CS Feed Pump 2 Flow Control
      _2090PU736I01AUTH1 : Bool := FALSE;   // Dont use Bit 1
      _2090PU736I01AUTH2 : Bool := FALSE;   // Dont use Bit 2
      _2090PU736I01AUTH3 : Bool := FALSE;   // Dont use Bit 3
      _2090PU736I01AUTH4 : Bool := FALSE;   // Dont use Bit 4
      _2090PU736I01AUTH5 : Bool := FALSE;   // Dont use Bit 5
      _2090PU736I01AUTH6 : Bool := FALSE;   // Dont use Bit 6
      _2090PU736I01AUTH7 : Bool := FALSE;   // Dont use Bit 7
      _2090PU620I01AUTH : Bool := FALSE;   // Carbon Pump Quench Tank Speed Control
      _2090PU620I01AUTH1 : Bool := FALSE;   // Dont use Bit 1
      _2090PU620I01AUTH2 : Bool := FALSE;   // Dont use Bit 2
      _2090PU620I01AUTH3 : Bool := FALSE;   // Dont use Bit 3
      _2090PU620I01AUTH4 : Bool := FALSE;   // Dont use Bit 4
      _2090PU620I01AUTH5 : Bool := FALSE;   // Dont use Bit 5
      _2090PU620I01AUTH6 : Bool := FALSE;   // Dont use Bit 6
      _2090PU620I01AUTH7 : Bool := FALSE;   // Dont use Bit 7
      _995CD100G04REQ04 : Bool := FALSE;   // Strip Process Finish Command
      _995CD100G04REQ041 : Bool := FALSE;   // Dont use Bit 1
      _995CD100G04REQ042 : Bool := FALSE;   // Dont use Bit 2
      _995CD100G04REQ043 : Bool := FALSE;   // Dont use Bit 3
      _995CD100G04REQ044 : Bool := FALSE;   // Dont use Bit 4
      _995CD100G04REQ045 : Bool := FALSE;   // Dont use Bit 5
      _995CD100G04REQ046 : Bool := FALSE;   // Dont use Bit 6
      _995CD100G04REQ047 : Bool := FALSE;   // Dont use Bit 7
      _995CD100G04REQ05 : Bool := FALSE;   // Strip Process Reset
      _995CD100G04REQ051 : Bool := FALSE;   // Dont use Bit 1
      _995CD100G04REQ052 : Bool := FALSE;   // Dont use Bit 2
      _995CD100G04REQ053 : Bool := FALSE;   // Dont use Bit 3
      _995CD100G04REQ054 : Bool := FALSE;   // Dont use Bit 4
      _995CD100G04REQ055 : Bool := FALSE;   // Dont use Bit 5
      _995CD100G04REQ056 : Bool := FALSE;   // Dont use Bit 6
      _995CD100G04REQ057 : Bool := FALSE;   // Dont use Bit 7
      _995CD100G04REQ06 : Bool := FALSE;   // ADR Command Reset All Strip Steps
      _995CD100G04REQ061 : Bool := FALSE;   // Dont use Bit 1
      _995CD100G04REQ062 : Bool := FALSE;   // Dont use Bit 2
      _995CD100G04REQ063 : Bool := FALSE;   // Dont use Bit 3
      _995CD100G04REQ064 : Bool := FALSE;   // Dont use Bit 4
      _995CD100G04REQ065 : Bool := FALSE;   // Dont use Bit 5
      _995CD100G04REQ066 : Bool := FALSE;   // Dont use Bit 6
      _995CD100G04REQ067 : Bool := FALSE;   // Dont use Bit 7
      _2090TK640Y08REQ01 : Bool := FALSE;   // Pressure Release Sequence
      _2090TK640Y08REQ011 : Bool := FALSE;   // Dont use Bit 1
      _2090TK640Y08REQ012 : Bool := FALSE;   // Dont use Bit 2
      _2090TK640Y08REQ013 : Bool := FALSE;   // Dont use Bit 3
      _2090TK640Y08REQ014 : Bool := FALSE;   // Dont use Bit 4
      _2090TK640Y08REQ015 : Bool := FALSE;   // Dont use Bit 5
      _2090TK640Y08REQ016 : Bool := FALSE;   // Dont use Bit 6
      _2090TK640Y08REQ017 : Bool := FALSE;   // Dont use Bit 7
      _2090TK641Y07REQ01 : Bool := FALSE;   // Pressure Release Sequence By Operator
      _2090TK641Y07REQ011 : Bool := FALSE;   // Dont use Bit 1
      _2090TK641Y07REQ012 : Bool := FALSE;   // Dont use Bit 2
      _2090TK641Y07REQ013 : Bool := FALSE;   // Dont use Bit 3
      _2090TK641Y07REQ014 : Bool := FALSE;   // Dont use Bit 4
      _2090TK641Y07REQ015 : Bool := FALSE;   // Dont use Bit 5
      _2090TK641Y07REQ016 : Bool := FALSE;   // Dont use Bit 6
      _2090TK641Y07REQ017 : Bool := FALSE;   // Dont use Bit 7
      _995CD100G04I12REQ01 : Bool := FALSE;   // Mix Sequence Start Command
      _995CD100G04I12REQ011 : Bool := FALSE;   // Dont use Bit 1
      _995CD100G04I12REQ012 : Bool := FALSE;   // Dont use Bit 2
      _995CD100G04I12REQ013 : Bool := FALSE;   // Dont use Bit 3
      _995CD100G04I12REQ014 : Bool := FALSE;   // Dont use Bit 4
      _995CD100G04I12REQ015 : Bool := FALSE;   // Dont use Bit 5
      _995CD100G04I12REQ016 : Bool := FALSE;   // Dont use Bit 6
      _995CD100G04I12REQ017 : Bool := FALSE;   // Dont use Bit 7
      _2090PU681I01AUTH : Bool := FALSE;   // Pump Strip Solution Speed Control
      _2090PU681I01AUTH1 : Bool := FALSE;   // Dont use Bit 1
      _2090PU681I01AUTH2 : Bool := FALSE;   // Dont use Bit 2
      _2090PU681I01AUTH3 : Bool := FALSE;   // Dont use Bit 3
      _2090PU681I01AUTH4 : Bool := FALSE;   // Dont use Bit 4
      _2090PU681I01AUTH5 : Bool := FALSE;   // Dont use Bit 5
      _2090PU681I01AUTH6 : Bool := FALSE;   // Dont use Bit 6
      _2090PU681I01AUTH7 : Bool := FALSE;   // Dont use Bit 7
      _2090PU682I01AUTH : Bool := FALSE;   // Pump Strip Solution Speed Control
      _2090PU682I01AUTH1 : Bool := FALSE;   // Dont use Bit 1
      _2090PU682I01AUTH2 : Bool := FALSE;   // Dont use Bit 2
      _2090PU682I01AUTH3 : Bool := FALSE;   // Dont use Bit 3
      _2090PU682I01AUTH4 : Bool := FALSE;   // Dont use Bit 4
      _2090PU682I01AUTH5 : Bool := FALSE;   // Dont use Bit 5
      _2090PU682I01AUTH6 : Bool := FALSE;   // Dont use Bit 6
      _2090PU682I01AUTH7 : Bool := FALSE;   // Dont use Bit 7
      _2090HT683I01AUTH : Bool := FALSE;   // Strip Solution Heater SCR-1 Temp Control
      _2090HT683I01AUTH1 : Bool := FALSE;   // Dont use Bit 1
      _2090HT683I01AUTH2 : Bool := FALSE;   // Dont use Bit 2
      _2090HT683I01AUTH3 : Bool := FALSE;   // Dont use Bit 3
      _2090HT683I01AUTH4 : Bool := FALSE;   // Dont use Bit 4
      _2090HT683I01AUTH5 : Bool := FALSE;   // Dont use Bit 5
      _2090HT683I01AUTH6 : Bool := FALSE;   // Dont use Bit 6
      _2090HT683I01AUTH7 : Bool := FALSE;   // Dont use Bit 7
      _2090HT684I01AUTH : Bool := FALSE;   // Strip Solution Heater SCR-2 Temp Control
      _2090HT684I01AUTH1 : Bool := FALSE;   // Dont use Bit 1
      _2090HT684I01AUTH2 : Bool := FALSE;   // Dont use Bit 2
      _2090HT684I01AUTH3 : Bool := FALSE;   // Dont use Bit 3
      _2090HT684I01AUTH4 : Bool := FALSE;   // Dont use Bit 4
      _2090HT684I01AUTH5 : Bool := FALSE;   // Dont use Bit 5
      _2090HT684I01AUTH6 : Bool := FALSE;   // Dont use Bit 6
      _2090HT684I01AUTH7 : Bool := FALSE;   // Dont use Bit 7
      _2090HT685I01AUTH : Bool := FALSE;   // Strip Solution Heater SCR-3 Temp Control
      _2090HT685I01AUTH1 : Bool := FALSE;   // Dont use Bit 1
      _2090HT685I01AUTH2 : Bool := FALSE;   // Dont use Bit 2
      _2090HT685I01AUTH3 : Bool := FALSE;   // Dont use Bit 3
      _2090HT685I01AUTH4 : Bool := FALSE;   // Dont use Bit 4
      _2090HT685I01AUTH5 : Bool := FALSE;   // Dont use Bit 5
      _2090HT685I01AUTH6 : Bool := FALSE;   // Dont use Bit 6
      _2090HT685I01AUTH7 : Bool := FALSE;   // Dont use Bit 7
      _995CD100G05REQ01 : Bool := FALSE;   // Acid Wash Process Stop
      _995CD100G05REQ011 : Bool := FALSE;   // Dont use Bit 1
      _995CD100G05REQ012 : Bool := FALSE;   // Dont use Bit 2
      _995CD100G05REQ013 : Bool := FALSE;   // Dont use Bit 3
      _995CD100G05REQ014 : Bool := FALSE;   // Dont use Bit 4
      _995CD100G05REQ015 : Bool := FALSE;   // Dont use Bit 5
      _995CD100G05REQ016 : Bool := FALSE;   // Dont use Bit 6
      _995CD100G05REQ017 : Bool := FALSE;   // Dont use Bit 7
      _995CD100G05REQ02 : Bool := FALSE;   // Pre Rinse Enable
      _995CD100G05REQ021 : Bool := FALSE;   // Dont use Bit 1
      _995CD100G05REQ022 : Bool := FALSE;   // Dont use Bit 2
      _995CD100G05REQ023 : Bool := FALSE;   // Dont use Bit 3
      _995CD100G05REQ024 : Bool := FALSE;   // Dont use Bit 4
      _995CD100G05REQ025 : Bool := FALSE;   // Dont use Bit 5
      _995CD100G05REQ026 : Bool := FALSE;   // Dont use Bit 6
      _995CD100G05REQ027 : Bool := FALSE;   // Dont use Bit 7
      _995CD100G05REQ03 : Bool := FALSE;   // Pre Rinse V2 Enable
      _995CD100G05REQ031 : Bool := FALSE;   // Dont use Bit 1
      _995CD100G05REQ032 : Bool := FALSE;   // Dont use Bit 2
      _995CD100G05REQ033 : Bool := FALSE;   // Dont use Bit 3
      _995CD100G05REQ034 : Bool := FALSE;   // Dont use Bit 4
      _995CD100G05REQ035 : Bool := FALSE;   // Dont use Bit 5
      _995CD100G05REQ036 : Bool := FALSE;   // Dont use Bit 6
      _995CD100G05REQ037 : Bool := FALSE;   // Dont use Bit 7
      _2090TK630Y09REQ01 : Bool := TRUE;   // TK630Y06 Drain Carbon Transfer
      _2090TK630Y09REQ011 : Bool := FALSE;   // Dont use Bit 1
      _2090TK630Y09REQ012 : Bool := FALSE;   // Dont use Bit 2
      _2090TK630Y09REQ013 : Bool := FALSE;   // Dont use Bit 3
      _2090TK630Y09REQ014 : Bool := FALSE;   // Dont use Bit 4
      _2090TK630Y09REQ015 : Bool := FALSE;   // Dont use Bit 5
      _2090TK630Y09REQ016 : Bool := FALSE;   // Dont use Bit 6
      _2090TK630Y09REQ017 : Bool := FALSE;   // Dont use Bit 7
      _995CD100G05I12REQ01 : Bool := FALSE;   // Acid Mix Initiated By Operator
      _995CD100G05I12REQ011 : Bool := FALSE;   // Dont use Bit 1
      _995CD100G05I12REQ012 : Bool := FALSE;   // Dont use Bit 2
      _995CD100G05I12REQ013 : Bool := FALSE;   // Dont use Bit 3
      _995CD100G05I12REQ014 : Bool := FALSE;   // Dont use Bit 4
      _995CD100G05I12REQ015 : Bool := FALSE;   // Dont use Bit 5
      _995CD100G05I12REQ016 : Bool := FALSE;   // Dont use Bit 6
      _995CD100G05I12REQ017 : Bool := FALSE;   // Dont use Bit 7
      _2095RC710A01I11AUTH : Bool := FALSE;   // Rectifier ADR, Current Setpoint
      _2095RC710A01I11AUTH1 : Bool := FALSE;   // Dont use Bit 1
      _2095RC710A01I11AUTH2 : Bool := FALSE;   // Dont use Bit 2
      _2095RC710A01I11AUTH3 : Bool := FALSE;   // Dont use Bit 3
      _2095RC710A01I11AUTH4 : Bool := FALSE;   // Dont use Bit 4
      _2095RC710A01I11AUTH5 : Bool := FALSE;   // Dont use Bit 5
      _2095RC710A01I11AUTH6 : Bool := FALSE;   // Dont use Bit 6
      _2095RC710A01I11AUTH7 : Bool := FALSE;   // Dont use Bit 7
      _2095RC710A01E11AUTH : Bool := FALSE;   // Rectifier ADR, Voltage Setpoint
      _2095RC710A01E11AUTH1 : Bool := FALSE;   // Dont use Bit 1
      _2095RC710A01E11AUTH2 : Bool := FALSE;   // Dont use Bit 2
      _2095RC710A01E11AUTH3 : Bool := FALSE;   // Dont use Bit 3
      _2095RC710A01E11AUTH4 : Bool := FALSE;   // Dont use Bit 4
      _2095RC710A01E11AUTH5 : Bool := FALSE;   // Dont use Bit 5
      _2095RC710A01E11AUTH6 : Bool := FALSE;   // Dont use Bit 6
      _2095RC710A01E11AUTH7 : Bool := FALSE;   // Dont use Bit 7
      _2095RC711A01I11AUTH : Bool := FALSE;   // Rectifier ADR, Current Setpoint
      _2095RC711A01I11AUTH1 : Bool := FALSE;   // Dont use Bit 1
      _2095RC711A01I11AUTH2 : Bool := FALSE;   // Dont use Bit 2
      _2095RC711A01I11AUTH3 : Bool := FALSE;   // Dont use Bit 3
      _2095RC711A01I11AUTH4 : Bool := FALSE;   // Dont use Bit 4
      _2095RC711A01I11AUTH5 : Bool := FALSE;   // Dont use Bit 5
      _2095RC711A01I11AUTH6 : Bool := FALSE;   // Dont use Bit 6
      _2095RC711A01I11AUTH7 : Bool := FALSE;   // Dont use Bit 7
      _2095RC711A01E11AUTH : Bool := FALSE;   // Rectifier ADR, Voltage Setpoint
      _2095RC711A01E11AUTH1 : Bool := FALSE;   // Dont use Bit 1
      _2095RC711A01E11AUTH2 : Bool := FALSE;   // Dont use Bit 2
      _2095RC711A01E11AUTH3 : Bool := FALSE;   // Dont use Bit 3
      _2095RC711A01E11AUTH4 : Bool := FALSE;   // Dont use Bit 4
      _2095RC711A01E11AUTH5 : Bool := FALSE;   // Dont use Bit 5
      _2095RC711A01E11AUTH6 : Bool := FALSE;   // Dont use Bit 6
      _2095RC711A01E11AUTH7 : Bool := FALSE;   // Dont use Bit 7
      _2095RC712A01I11AUTH : Bool := FALSE;   // Rectifier ADR, Current Setpoint
      _2095RC712A01I11AUTH1 : Bool := FALSE;   // Dont use Bit 1
      _2095RC712A01I11AUTH2 : Bool := FALSE;   // Dont use Bit 2
      _2095RC712A01I11AUTH3 : Bool := FALSE;   // Dont use Bit 3
      _2095RC712A01I11AUTH4 : Bool := FALSE;   // Dont use Bit 4
      _2095RC712A01I11AUTH5 : Bool := FALSE;   // Dont use Bit 5
      _2095RC712A01I11AUTH6 : Bool := FALSE;   // Dont use Bit 6
      _2095RC712A01I11AUTH7 : Bool := FALSE;   // Dont use Bit 7
      _2095RC712A01E11AUTH : Bool := FALSE;   // Rectifier ADR, Voltage Setpoint
      _2095RC712A01E11AUTH1 : Bool := FALSE;   // Dont use Bit 1
      _2095RC712A01E11AUTH2 : Bool := FALSE;   // Dont use Bit 2
      _2095RC712A01E11AUTH3 : Bool := FALSE;   // Dont use Bit 3
      _2095RC712A01E11AUTH4 : Bool := FALSE;   // Dont use Bit 4
      _2095RC712A01E11AUTH5 : Bool := FALSE;   // Dont use Bit 5
      _2095RC712A01E11AUTH6 : Bool := FALSE;   // Dont use Bit 6
      _2095RC712A01E11AUTH7 : Bool := FALSE;   // Dont use Bit 7
      _2095RC713A01I11AUTH : Bool := FALSE;   // Rectifier ADR, Current Setpoint
      _2095RC713A01I11AUTH1 : Bool := FALSE;   // Dont use Bit 1
      _2095RC713A01I11AUTH2 : Bool := FALSE;   // Dont use Bit 2
      _2095RC713A01I11AUTH3 : Bool := FALSE;   // Dont use Bit 3
      _2095RC713A01I11AUTH4 : Bool := FALSE;   // Dont use Bit 4
      _2095RC713A01I11AUTH5 : Bool := FALSE;   // Dont use Bit 5
      _2095RC713A01I11AUTH6 : Bool := FALSE;   // Dont use Bit 6
      _2095RC713A01I11AUTH7 : Bool := FALSE;   // Dont use Bit 7
      _2095RC713A01E11AUTH : Bool := FALSE;   // Rectifier ADR, Voltage Setpoint
      _2095RC713A01E11AUTH1 : Bool := FALSE;   // Dont use Bit 1
      _2095RC713A01E11AUTH2 : Bool := FALSE;   // Dont use Bit 2
      _2095RC713A01E11AUTH3 : Bool := FALSE;   // Dont use Bit 3
      _2095RC713A01E11AUTH4 : Bool := FALSE;   // Dont use Bit 4
      _2095RC713A01E11AUTH5 : Bool := FALSE;   // Dont use Bit 5
      _2095RC713A01E11AUTH6 : Bool := FALSE;   // Dont use Bit 6
      _2095RC713A01E11AUTH7 : Bool := FALSE;   // Dont use Bit 7
      _2095RC714A01I11AUTH : Bool := FALSE;   // Rectifier ADR, Current Setpoint
      _2095RC714A01I11AUTH1 : Bool := FALSE;   // Dont use Bit 1
      _2095RC714A01I11AUTH2 : Bool := FALSE;   // Dont use Bit 2
      _2095RC714A01I11AUTH3 : Bool := FALSE;   // Dont use Bit 3
      _2095RC714A01I11AUTH4 : Bool := FALSE;   // Dont use Bit 4
      _2095RC714A01I11AUTH5 : Bool := FALSE;   // Dont use Bit 5
      _2095RC714A01I11AUTH6 : Bool := FALSE;   // Dont use Bit 6
      _2095RC714A01I11AUTH7 : Bool := FALSE;   // Dont use Bit 7
      _2095RC714A01E11AUTH : Bool := FALSE;   // Rectifier ADR, Voltage Setpoint
      _2095RC714A01E11AUTH1 : Bool := FALSE;   // Dont use Bit 1
      _2095RC714A01E11AUTH2 : Bool := FALSE;   // Dont use Bit 2
      _2095RC714A01E11AUTH3 : Bool := FALSE;   // Dont use Bit 3
      _2095RC714A01E11AUTH4 : Bool := FALSE;   // Dont use Bit 4
      _2095RC714A01E11AUTH5 : Bool := FALSE;   // Dont use Bit 5
      _2095RC714A01E11AUTH6 : Bool := FALSE;   // Dont use Bit 6
      _2095RC714A01E11AUTH7 : Bool := FALSE;   // Dont use Bit 7
      _995CS100_PID01AUTH : Bool := FALSE;   // PID01
      _995CS100_PID01AUTH1 : Bool := FALSE;   // Dont use Bit 1
      _995CS100_PID01AUTH2 : Bool := FALSE;   // Dont use Bit 2
      _995CS100_PID01AUTH3 : Bool := FALSE;   // Dont use Bit 3
      _995CS100_PID01AUTH4 : Bool := FALSE;   // Dont use Bit 4
      _995CS100_PID01AUTH5 : Bool := FALSE;   // Dont use Bit 5
      _995CS100_PID01AUTH6 : Bool := FALSE;   // Dont use Bit 6
      _995CS100_PID01AUTH7 : Bool := FALSE;   // Dont use Bit 7
      _995CS100_PID02AUTH : Bool := FALSE;   // PID02
      _995CS100_PID02AUTH1 : Bool := FALSE;   // Dont use Bit 1
      _995CS100_PID02AUTH2 : Bool := FALSE;   // Dont use Bit 2
      _995CS100_PID02AUTH3 : Bool := FALSE;   // Dont use Bit 3
      _995CS100_PID02AUTH4 : Bool := FALSE;   // Dont use Bit 4
      _995CS100_PID02AUTH5 : Bool := FALSE;   // Dont use Bit 5
      _995CS100_PID02AUTH6 : Bool := FALSE;   // Dont use Bit 6
      _995CS100_PID02AUTH7 : Bool := FALSE;   // Dont use Bit 7
      _995CS100_PID03AUTH : Bool := FALSE;   // PID03
      _995CS100_PID03AUTH1 : Bool := FALSE;   // Dont use Bit 1
      _995CS100_PID03AUTH2 : Bool := FALSE;   // Dont use Bit 2
      _995CS100_PID03AUTH3 : Bool := FALSE;   // Dont use Bit 3
      _995CS100_PID03AUTH4 : Bool := FALSE;   // Dont use Bit 4
      _995CS100_PID03AUTH5 : Bool := FALSE;   // Dont use Bit 5
      _995CS100_PID03AUTH6 : Bool := FALSE;   // Dont use Bit 6
      _995CS100_PID03AUTH7 : Bool := FALSE;   // Dont use Bit 7
      _995CS100_PID04AUTH : Bool := FALSE;   // PID04
      _995CS100_PID04AUTH1 : Bool := FALSE;   // Dont use Bit 1
      _995CS100_PID04AUTH2 : Bool := FALSE;   // Dont use Bit 2
      _995CS100_PID04AUTH3 : Bool := FALSE;   // Dont use Bit 3
      _995CS100_PID04AUTH4 : Bool := FALSE;   // Dont use Bit 4
      _995CS100_PID04AUTH5 : Bool := FALSE;   // Dont use Bit 5
      _995CS100_PID04AUTH6 : Bool := FALSE;   // Dont use Bit 6
      _995CS100_PID04AUTH7 : Bool := FALSE;   // Dont use Bit 7
      _995CS100_PID05AUTH : Bool := FALSE;   // PID05
      _995CS100_PID05AUTH1 : Bool := FALSE;   // Dont use Bit 1
      _995CS100_PID05AUTH2 : Bool := FALSE;   // Dont use Bit 2
      _995CS100_PID05AUTH3 : Bool := FALSE;   // Dont use Bit 3
      _995CS100_PID05AUTH4 : Bool := FALSE;   // Dont use Bit 4
      _995CS100_PID05AUTH5 : Bool := FALSE;   // Dont use Bit 5
      _995CS100_PID05AUTH6 : Bool := FALSE;   // Dont use Bit 6
      _995CS100_PID05AUTH7 : Bool := FALSE;   // Dont use Bit 7
      _995CS100_PID06AUTH : Bool := FALSE;   // PID06
      _995CS100_PID06AUTH1 : Bool := FALSE;   // Dont use Bit 1
      _995CS100_PID06AUTH2 : Bool := FALSE;   // Dont use Bit 2
      _995CS100_PID06AUTH3 : Bool := FALSE;   // Dont use Bit 3
      _995CS100_PID06AUTH4 : Bool := FALSE;   // Dont use Bit 4
      _995CS100_PID06AUTH5 : Bool := FALSE;   // Dont use Bit 5
      _995CS100_PID06AUTH6 : Bool := FALSE;   // Dont use Bit 6
      _995CS100_PID06AUTH7 : Bool := FALSE;   // Dont use Bit 7
      _995CS100_PID07AUTH : Bool := FALSE;   // PID07
      _995CS100_PID07AUTH1 : Bool := FALSE;   // Dont use Bit 1
      _995CS100_PID07AUTH2 : Bool := FALSE;   // Dont use Bit 2
      _995CS100_PID07AUTH3 : Bool := FALSE;   // Dont use Bit 3
      _995CS100_PID07AUTH4 : Bool := FALSE;   // Dont use Bit 4
      _995CS100_PID07AUTH5 : Bool := FALSE;   // Dont use Bit 5
      _995CS100_PID07AUTH6 : Bool := FALSE;   // Dont use Bit 6
      _995CS100_PID07AUTH7 : Bool := FALSE;   // Dont use Bit 7
      _995CS100_PID08AUTH : Bool := FALSE;   // PID08
      _995CS100_PID08AUTH1 : Bool := FALSE;   // Dont use Bit 1
      _995CS100_PID08AUTH2 : Bool := FALSE;   // Dont use Bit 2
      _995CS100_PID08AUTH3 : Bool := FALSE;   // Dont use Bit 3
      _995CS100_PID08AUTH4 : Bool := FALSE;   // Dont use Bit 4
      _995CS100_PID08AUTH5 : Bool := FALSE;   // Dont use Bit 5
      _995CS100_PID08AUTH6 : Bool := FALSE;   // Dont use Bit 6
      _995CS100_PID08AUTH7 : Bool := FALSE;   // Dont use Bit 7
      _995CS100_PID09AUTH : Bool := FALSE;   // PID09
      _995CS100_PID09AUTH1 : Bool := FALSE;   // Dont use Bit 1
      _995CS100_PID09AUTH2 : Bool := FALSE;   // Dont use Bit 2
      _995CS100_PID09AUTH3 : Bool := FALSE;   // Dont use Bit 3
      _995CS100_PID09AUTH4 : Bool := FALSE;   // Dont use Bit 4
      _995CS100_PID09AUTH5 : Bool := FALSE;   // Dont use Bit 5
      _995CS100_PID09AUTH6 : Bool := FALSE;   // Dont use Bit 6
      _995CS100_PID09AUTH7 : Bool := FALSE;   // Dont use Bit 7
      _995CS100_PID10AUTH : Bool := FALSE;   // PID10
      _995CS100_PID10AUTH1 : Bool := FALSE;   // Dont use Bit 1
      _995CS100_PID10AUTH2 : Bool := FALSE;   // Dont use Bit 2
      _995CS100_PID10AUTH3 : Bool := FALSE;   // Dont use Bit 3
      _995CS100_PID10AUTH4 : Bool := FALSE;   // Dont use Bit 4
      _995CS100_PID10AUTH5 : Bool := FALSE;   // Dont use Bit 5
      _995CS100_PID10AUTH6 : Bool := FALSE;   // Dont use Bit 6
      _995CS100_PID10AUTH7 : Bool := FALSE;   // Dont use Bit 7
      _995CS100_PID11AUTH : Bool := FALSE;   // PID11
      _995CS100_PID11AUTH1 : Bool := FALSE;   // Dont use Bit 1
      _995CS100_PID11AUTH2 : Bool := FALSE;   // Dont use Bit 2
      _995CS100_PID11AUTH3 : Bool := FALSE;   // Dont use Bit 3
      _995CS100_PID11AUTH4 : Bool := FALSE;   // Dont use Bit 4
      _995CS100_PID11AUTH5 : Bool := FALSE;   // Dont use Bit 5
      _995CS100_PID11AUTH6 : Bool := FALSE;   // Dont use Bit 6
      _995CS100_PID11AUTH7 : Bool := FALSE;   // Dont use Bit 7
      _995CS100_PID12AUTH : Bool := FALSE;   // PID12
      _995CS100_PID12AUTH1 : Bool := FALSE;   // Dont use Bit 1
      _995CS100_PID12AUTH2 : Bool := FALSE;   // Dont use Bit 2
      _995CS100_PID12AUTH3 : Bool := FALSE;   // Dont use Bit 3
      _995CS100_PID12AUTH4 : Bool := FALSE;   // Dont use Bit 4
      _995CS100_PID12AUTH5 : Bool := FALSE;   // Dont use Bit 5
      _995CS100_PID12AUTH6 : Bool := FALSE;   // Dont use Bit 6
      _995CS100_PID12AUTH7 : Bool := FALSE;   // Dont use Bit 7
      _995CS100_PID13AUTH : Bool := FALSE;   // PID13
      _995CS100_PID13AUTH1 : Bool := FALSE;   // Dont use Bit 1
      _995CS100_PID13AUTH2 : Bool := FALSE;   // Dont use Bit 2
      _995CS100_PID13AUTH3 : Bool := FALSE;   // Dont use Bit 3
      _995CS100_PID13AUTH4 : Bool := FALSE;   // Dont use Bit 4
      _995CS100_PID13AUTH5 : Bool := FALSE;   // Dont use Bit 5
      _995CS100_PID13AUTH6 : Bool := FALSE;   // Dont use Bit 6
      _995CS100_PID13AUTH7 : Bool := FALSE;   // Dont use Bit 7
      _995CS100_PID14AUTH : Bool := FALSE;   // PID14
      _995CS100_PID14AUTH1 : Bool := FALSE;   // Dont use Bit 1
      _995CS100_PID14AUTH2 : Bool := FALSE;   // Dont use Bit 2
      _995CS100_PID14AUTH3 : Bool := FALSE;   // Dont use Bit 3
      _995CS100_PID14AUTH4 : Bool := FALSE;   // Dont use Bit 4
      _995CS100_PID14AUTH5 : Bool := FALSE;   // Dont use Bit 5
      _995CS100_PID14AUTH6 : Bool := FALSE;   // Dont use Bit 6
      _995CS100_PID14AUTH7 : Bool := FALSE;   // Dont use Bit 7
      _995CS100_PID15AUTH : Bool := FALSE;   // PID15
      _995CS100_PID15AUTH1 : Bool := FALSE;   // Dont use Bit 1
      _995CS100_PID15AUTH2 : Bool := FALSE;   // Dont use Bit 2
      _995CS100_PID15AUTH3 : Bool := FALSE;   // Dont use Bit 3
      _995CS100_PID15AUTH4 : Bool := FALSE;   // Dont use Bit 4
      _995CS100_PID15AUTH5 : Bool := FALSE;   // Dont use Bit 5
      _995CS100_PID15AUTH6 : Bool := FALSE;   // Dont use Bit 6
      _995CS100_PID15AUTH7 : Bool := FALSE;   // Dont use Bit 7
      _995CS100_SIMPLEREQ01 : Bool := FALSE;   // SIMPLEREQ01
      _995CS100_SIMPLEREQ011 : Bool := FALSE;   // Dont use Bit 1
      _995CS100_SIMPLEREQ012 : Bool := FALSE;   // Dont use Bit 2
      _995CS100_SIMPLEREQ013 : Bool := FALSE;   // Dont use Bit 3
      _995CS100_SIMPLEREQ014 : Bool := FALSE;   // Dont use Bit 4
      _995CS100_SIMPLEREQ015 : Bool := FALSE;   // Dont use Bit 5
      _995CS100_SIMPLEREQ016 : Bool := FALSE;   // Dont use Bit 6
      _995CS100_SIMPLEREQ017 : Bool := FALSE;   // Dont use Bit 7
      _995CS100_SIMPLEREQ02 : Bool := FALSE;   // SIMPLEREQ02
      _995CS100_SIMPLEREQ021 : Bool := FALSE;   // Dont use Bit 1
      _995CS100_SIMPLEREQ022 : Bool := FALSE;   // Dont use Bit 2
      _995CS100_SIMPLEREQ023 : Bool := FALSE;   // Dont use Bit 3
      _995CS100_SIMPLEREQ024 : Bool := FALSE;   // Dont use Bit 4
      _995CS100_SIMPLEREQ025 : Bool := FALSE;   // Dont use Bit 5
      _995CS100_SIMPLEREQ026 : Bool := FALSE;   // Dont use Bit 6
      _995CS100_SIMPLEREQ027 : Bool := FALSE;   // Dont use Bit 7
      _995CS100_SIMPLEREQ03 : Bool := FALSE;   // SIMPLEREQ03
      _995CS100_SIMPLEREQ031 : Bool := FALSE;   // Dont use Bit 1
      _995CS100_SIMPLEREQ032 : Bool := FALSE;   // Dont use Bit 2
      _995CS100_SIMPLEREQ033 : Bool := FALSE;   // Dont use Bit 3
      _995CS100_SIMPLEREQ034 : Bool := FALSE;   // Dont use Bit 4
      _995CS100_SIMPLEREQ035 : Bool := FALSE;   // Dont use Bit 5
      _995CS100_SIMPLEREQ036 : Bool := FALSE;   // Dont use Bit 6
      _995CS100_SIMPLEREQ037 : Bool := FALSE;   // Dont use Bit 7
      _995CS100_SIMPLEREQ04 : Bool := FALSE;   // SIMPLEREQ04
      _995CS100_SIMPLEREQ041 : Bool := FALSE;   // Dont use Bit 1
      _995CS100_SIMPLEREQ042 : Bool := FALSE;   // Dont use Bit 2
      _995CS100_SIMPLEREQ043 : Bool := FALSE;   // Dont use Bit 3
      _995CS100_SIMPLEREQ044 : Bool := FALSE;   // Dont use Bit 4
      _995CS100_SIMPLEREQ045 : Bool := FALSE;   // Dont use Bit 5
      _995CS100_SIMPLEREQ046 : Bool := FALSE;   // Dont use Bit 6
      _995CS100_SIMPLEREQ047 : Bool := FALSE;   // Dont use Bit 7
      _995CS100_SIMPLEREQ05 : Bool := FALSE;   // SIMPLEREQ05
      _995CS100_SIMPLEREQ051 : Bool := FALSE;   // Dont use Bit 1
      _995CS100_SIMPLEREQ052 : Bool := FALSE;   // Dont use Bit 2
      _995CS100_SIMPLEREQ053 : Bool := FALSE;   // Dont use Bit 3
      _995CS100_SIMPLEREQ054 : Bool := FALSE;   // Dont use Bit 4
      _995CS100_SIMPLEREQ055 : Bool := FALSE;   // Dont use Bit 5
      _995CS100_SIMPLEREQ056 : Bool := FALSE;   // Dont use Bit 6
      _995CS100_SIMPLEREQ057 : Bool := FALSE;   // Dont use Bit 7
      _995CS100_SIMPLEREQ06 : Bool := FALSE;   // SIMPLEREQ06
      _995CS100_SIMPLEREQ061 : Bool := FALSE;   // Dont use Bit 1
      _995CS100_SIMPLEREQ062 : Bool := FALSE;   // Dont use Bit 2
      _995CS100_SIMPLEREQ063 : Bool := FALSE;   // Dont use Bit 3
      _995CS100_SIMPLEREQ064 : Bool := FALSE;   // Dont use Bit 4
      _995CS100_SIMPLEREQ065 : Bool := FALSE;   // Dont use Bit 5
      _995CS100_SIMPLEREQ066 : Bool := FALSE;   // Dont use Bit 6
      _995CS100_SIMPLEREQ067 : Bool := FALSE;   // Dont use Bit 7
      _995CS100_SIMPLEREQ07 : Bool := FALSE;   // SIMPLEREQ07
      _995CS100_SIMPLEREQ071 : Bool := FALSE;   // Dont use Bit 1
      _995CS100_SIMPLEREQ072 : Bool := FALSE;   // Dont use Bit 2
      _995CS100_SIMPLEREQ073 : Bool := FALSE;   // Dont use Bit 3
      _995CS100_SIMPLEREQ074 : Bool := FALSE;   // Dont use Bit 4
      _995CS100_SIMPLEREQ075 : Bool := FALSE;   // Dont use Bit 5
      _995CS100_SIMPLEREQ076 : Bool := FALSE;   // Dont use Bit 6
      _995CS100_SIMPLEREQ077 : Bool := FALSE;   // Dont use Bit 7
      _995CS100_SIMPLEREQ08 : Bool := FALSE;   // SIMPLEREQ08
      _995CS100_SIMPLEREQ081 : Bool := FALSE;   // Dont use Bit 1
      _995CS100_SIMPLEREQ082 : Bool := FALSE;   // Dont use Bit 2
      _995CS100_SIMPLEREQ083 : Bool := FALSE;   // Dont use Bit 3
      _995CS100_SIMPLEREQ084 : Bool := FALSE;   // Dont use Bit 4
      _995CS100_SIMPLEREQ085 : Bool := FALSE;   // Dont use Bit 5
      _995CS100_SIMPLEREQ086 : Bool := FALSE;   // Dont use Bit 6
      _995CS100_SIMPLEREQ087 : Bool := FALSE;   // Dont use Bit 7
      _995CS100_SIMPLEREQ09 : Bool := FALSE;   // SIMPLEREQ09
      _995CS100_SIMPLEREQ091 : Bool := FALSE;   // Dont use Bit 1
      _995CS100_SIMPLEREQ092 : Bool := FALSE;   // Dont use Bit 2
      _995CS100_SIMPLEREQ093 : Bool := FALSE;   // Dont use Bit 3
      _995CS100_SIMPLEREQ094 : Bool := FALSE;   // Dont use Bit 4
      _995CS100_SIMPLEREQ095 : Bool := FALSE;   // Dont use Bit 5
      _995CS100_SIMPLEREQ096 : Bool := FALSE;   // Dont use Bit 6
      _995CS100_SIMPLEREQ097 : Bool := FALSE;   // Dont use Bit 7
      _995CS100_SIMPLEREQ10 : Bool := FALSE;   // SIMPLEREQ10
      _995CS100_SIMPLEREQ101 : Bool := FALSE;   // Dont use Bit 1
      _995CS100_SIMPLEREQ102 : Bool := FALSE;   // Dont use Bit 2
      _995CS100_SIMPLEREQ103 : Bool := FALSE;   // Dont use Bit 3
      _995CS100_SIMPLEREQ104 : Bool := FALSE;   // Dont use Bit 4
      _995CS100_SIMPLEREQ105 : Bool := FALSE;   // Dont use Bit 5
      _995CS100_SIMPLEREQ106 : Bool := FALSE;   // Dont use Bit 6
      _995CS100_SIMPLEREQ107 : Bool := FALSE;   // Dont use Bit 7
      _995CS100_SIMPLEREQ11 : Bool := FALSE;   // SIMPLEREQ11
      _995CS100_SIMPLEREQ111 : Bool := FALSE;   // Dont use Bit 1
      _995CS100_SIMPLEREQ112 : Bool := FALSE;   // Dont use Bit 2
      _995CS100_SIMPLEREQ113 : Bool := FALSE;   // Dont use Bit 3
      _995CS100_SIMPLEREQ114 : Bool := FALSE;   // Dont use Bit 4
      _995CS100_SIMPLEREQ115 : Bool := FALSE;   // Dont use Bit 5
      _995CS100_SIMPLEREQ116 : Bool := FALSE;   // Dont use Bit 6
      _995CS100_SIMPLEREQ117 : Bool := FALSE;   // Dont use Bit 7
      _995CS100_SIMPLEREQ12 : Bool := FALSE;   // SIMPLEREQ12
      _995CS100_SIMPLEREQ121 : Bool := FALSE;   // Dont use Bit 1
      _995CS100_SIMPLEREQ122 : Bool := FALSE;   // Dont use Bit 2
      _995CS100_SIMPLEREQ123 : Bool := FALSE;   // Dont use Bit 3
      _995CS100_SIMPLEREQ124 : Bool := FALSE;   // Dont use Bit 4
      _995CS100_SIMPLEREQ125 : Bool := FALSE;   // Dont use Bit 5
      _995CS100_SIMPLEREQ126 : Bool := FALSE;   // Dont use Bit 6
      _995CS100_SIMPLEREQ127 : Bool := FALSE;   // Dont use Bit 7
      _995CS100_SIMPLEREQ13 : Bool := FALSE;   // SIMPLEREQ13
      _995CS100_SIMPLEREQ131 : Bool := FALSE;   // Dont use Bit 1
      _995CS100_SIMPLEREQ132 : Bool := FALSE;   // Dont use Bit 2
      _995CS100_SIMPLEREQ133 : Bool := FALSE;   // Dont use Bit 3
      _995CS100_SIMPLEREQ134 : Bool := FALSE;   // Dont use Bit 4
      _995CS100_SIMPLEREQ135 : Bool := FALSE;   // Dont use Bit 5
      _995CS100_SIMPLEREQ136 : Bool := FALSE;   // Dont use Bit 6
      _995CS100_SIMPLEREQ137 : Bool := FALSE;   // Dont use Bit 7
      _995CS100_SIMPLEREQ14 : Bool := FALSE;   // SIMPLEREQ14
      _995CS100_SIMPLEREQ141 : Bool := FALSE;   // Dont use Bit 1
      _995CS100_SIMPLEREQ142 : Bool := FALSE;   // Dont use Bit 2
      _995CS100_SIMPLEREQ143 : Bool := FALSE;   // Dont use Bit 3
      _995CS100_SIMPLEREQ144 : Bool := FALSE;   // Dont use Bit 4
      _995CS100_SIMPLEREQ145 : Bool := FALSE;   // Dont use Bit 5
      _995CS100_SIMPLEREQ146 : Bool := FALSE;   // Dont use Bit 6
      _995CS100_SIMPLEREQ147 : Bool := FALSE;   // Dont use Bit 7
      _995CS100_SIMPLEREQ15 : Bool := FALSE;   // SIMPLEREQ15
      _995CS100_SIMPLEREQ151 : Bool := FALSE;   // Dont use Bit 1
      _995CS100_SIMPLEREQ152 : Bool := FALSE;   // Dont use Bit 2
      _995CS100_SIMPLEREQ153 : Bool := FALSE;   // Dont use Bit 3
      _995CS100_SIMPLEREQ154 : Bool := FALSE;   // Dont use Bit 4
      _995CS100_SIMPLEREQ155 : Bool := FALSE;   // Dont use Bit 5
      _995CS100_SIMPLEREQ156 : Bool := FALSE;   // Dont use Bit 6
      _995CS100_SIMPLEREQ157 : Bool := FALSE;   // Dont use Bit 7
      _995CS100_SIMPLEREQ16 : Bool := FALSE;   // SIMPLEREQ16
      _995CS100_SIMPLEREQ161 : Bool := FALSE;   // Dont use Bit 1
      _995CS100_SIMPLEREQ162 : Bool := FALSE;   // Dont use Bit 2
      _995CS100_SIMPLEREQ163 : Bool := FALSE;   // Dont use Bit 3
      _995CS100_SIMPLEREQ164 : Bool := FALSE;   // Dont use Bit 4
      _995CS100_SIMPLEREQ165 : Bool := FALSE;   // Dont use Bit 5
      _995CS100_SIMPLEREQ166 : Bool := FALSE;   // Dont use Bit 6
      _995CS100_SIMPLEREQ167 : Bool := FALSE;   // Dont use Bit 7
      _995CS100_SIMPLEREQ17 : Bool := FALSE;   // SIMPLEREQ17
      _995CS100_SIMPLEREQ171 : Bool := FALSE;   // Dont use Bit 1
      _995CS100_SIMPLEREQ172 : Bool := FALSE;   // Dont use Bit 2
      _995CS100_SIMPLEREQ173 : Bool := FALSE;   // Dont use Bit 3
      _995CS100_SIMPLEREQ174 : Bool := FALSE;   // Dont use Bit 4
      _995CS100_SIMPLEREQ175 : Bool := FALSE;   // Dont use Bit 5
      _995CS100_SIMPLEREQ176 : Bool := FALSE;   // Dont use Bit 6
      _995CS100_SIMPLEREQ177 : Bool := FALSE;   // Dont use Bit 7
      _995CS100_SIMPLEREQ18 : Bool := FALSE;   // SIMPLEREQ18
      _995CS100_SIMPLEREQ181 : Bool := FALSE;   // Dont use Bit 1
      _995CS100_SIMPLEREQ182 : Bool := FALSE;   // Dont use Bit 2
      _995CS100_SIMPLEREQ183 : Bool := FALSE;   // Dont use Bit 3
      _995CS100_SIMPLEREQ184 : Bool := FALSE;   // Dont use Bit 4
      _995CS100_SIMPLEREQ185 : Bool := FALSE;   // Dont use Bit 5
      _995CS100_SIMPLEREQ186 : Bool := FALSE;   // Dont use Bit 6
      _995CS100_SIMPLEREQ187 : Bool := FALSE;   // Dont use Bit 7
      _995CS100_SIMPLEREQ19 : Bool := FALSE;   // SIMPLEREQ19
      _995CS100_SIMPLEREQ191 : Bool := FALSE;   // Dont use Bit 1
      _995CS100_SIMPLEREQ192 : Bool := FALSE;   // Dont use Bit 2
      _995CS100_SIMPLEREQ193 : Bool := FALSE;   // Dont use Bit 3
      _995CS100_SIMPLEREQ194 : Bool := FALSE;   // Dont use Bit 4
      _995CS100_SIMPLEREQ195 : Bool := FALSE;   // Dont use Bit 5
      _995CS100_SIMPLEREQ196 : Bool := FALSE;   // Dont use Bit 6
      _995CS100_SIMPLEREQ197 : Bool := FALSE;   // Dont use Bit 7
      _995CS100_SIMPLEREQ20 : Bool := FALSE;   // SIMPLEREQ20
      _995CS100_SIMPLEREQ201 : Bool := FALSE;   // Dont use Bit 1
      _995CS100_SIMPLEREQ202 : Bool := FALSE;   // Dont use Bit 2
      _995CS100_SIMPLEREQ203 : Bool := FALSE;   // Dont use Bit 3
      _995CS100_SIMPLEREQ204 : Bool := FALSE;   // Dont use Bit 4
      _995CS100_SIMPLEREQ205 : Bool := FALSE;   // Dont use Bit 5
      _995CS100_SIMPLEREQ206 : Bool := FALSE;   // Dont use Bit 6
      _995CS100_SIMPLEREQ207 : Bool := FALSE;   // Dont use Bit 7
   END_VAR
BEGIN
END_DATA_BLOCK

DATA_BLOCK "ACESYS_HMI_PID_SPA"   // DB15
TITLE = ACESYS PID SPA DB
{ S7_Optimized_Access := 'FALSE' }
AUTHOR : METIS
FAMILY : ACESYS
NAME : PID_SP
VERSION : 8.0
   VAR
      PID : Array[0..100] of Struct   // Setpoint AUTO from HMI
         SP : Real;   // Auto Setpoint Eng. Units
      END_STRUCT;
   END_VAR
BEGIN
   PID[0].SP := 0.0;
   PID[1].SP := 6.388889;
   PID[2].SP := 6.388888;
   PID[3].SP := 0.0;
   PID[4].SP := 7.398004;
   PID[5].SP := 7.398004;
   PID[6].SP := 0.07957175;
   PID[7].SP := 0.0;
   PID[8].SP := 0.0;
   PID[9].SP := 0.0;
   PID[10].SP := 0.0;
   PID[11].SP := 1.566117;
   PID[12].SP := 0.0;
   PID[13].SP := 1.388889;
   PID[14].SP := 0.0;
   PID[15].SP := 0.0;
   PID[16].SP := 0.0;
   PID[17].SP := 0.0;
   PID[18].SP := 0.0;
   PID[19].SP := 0.0;
   PID[20].SP := 0.0;
   PID[21].SP := 0.0;
   PID[22].SP := 0.0;
   PID[23].SP := 0.0;
   PID[24].SP := 0.0;
   PID[25].SP := 0.0;
   PID[26].SP := 0.0;
   PID[27].SP := 0.0;
   PID[28].SP := 0.0;
   PID[29].SP := 0.0;
   PID[30].SP := 0.0;
   PID[31].SP := 0.0;
   PID[32].SP := 0.0;
   PID[33].SP := 0.0;
   PID[34].SP := 0.0;
   PID[35].SP := 0.0;
   PID[36].SP := 0.0;
   PID[37].SP := 0.0;
   PID[38].SP := 0.0;
   PID[39].SP := 0.0;
   PID[40].SP := 0.0;
   PID[41].SP := 0.0;
   PID[42].SP := 0.0;
   PID[43].SP := 0.0;
   PID[44].SP := 0.0;
   PID[45].SP := 0.0;
   PID[46].SP := 0.0;
   PID[47].SP := 0.0;
   PID[48].SP := 0.0;
   PID[49].SP := 0.0;
   PID[50].SP := 0.0;
   PID[51].SP := 0.0;
   PID[52].SP := 0.0;
   PID[53].SP := 0.0;
   PID[54].SP := 0.0;
   PID[55].SP := 60.0;
   PID[56].SP := 0.0;
   PID[57].SP := 0.0;
   PID[58].SP := 0.0;
   PID[59].SP := 0.0;
   PID[60].SP := 0.0;
   PID[61].SP := 0.0;
   PID[62].SP := 0.0;
   PID[63].SP := 0.0;
   PID[64].SP := 0.0;
   PID[65].SP := 0.0;
   PID[66].SP := 0.0;
   PID[67].SP := 0.0;
   PID[68].SP := 0.0;
   PID[69].SP := 0.0;
   PID[70].SP := 0.0;
   PID[71].SP := 0.0;
   PID[72].SP := 0.0;
   PID[73].SP := 0.0;
   PID[74].SP := 0.0;
   PID[75].SP := 0.0;
   PID[76].SP := 0.0;
   PID[77].SP := 0.0;
   PID[78].SP := 0.0;
   PID[79].SP := 0.0;
   PID[80].SP := 0.0;
   PID[81].SP := 0.0;
   PID[82].SP := 0.0;
   PID[83].SP := 0.0;
   PID[84].SP := 0.0;
   PID[85].SP := 0.0;
   PID[86].SP := 0.0;
   PID[87].SP := 0.0;
   PID[88].SP := 0.0;
   PID[89].SP := 0.0;
   PID[90].SP := 0.0;
   PID[91].SP := 0.0;
   PID[92].SP := 0.0;
   PID[93].SP := 0.0;
   PID[94].SP := 0.0;
   PID[95].SP := 0.0;
   PID[96].SP := 0.0;
   PID[97].SP := 0.0;
   PID[98].SP := 0.0;
   PID[99].SP := 0.0;
   PID[100].SP := 0.0;
END_DATA_BLOCK

DATA_BLOCK "ACESYS_HMI_PID_SPM"   // DB16
TITLE = ACESYS PID SPM DB
{ S7_Optimized_Access := 'FALSE' }
AUTHOR : METIS
FAMILY : ACESYS
NAME : PID_SP
VERSION : 8.0
   VAR
      PID : Array[0..100] of Struct   // Setpoint MAN from HMI
         SP : Real;   // MANUAL Setpoint in Pct
      END_STRUCT;
   END_VAR
BEGIN
   PID[0].SP := 0.0;
   PID[1].SP := 100.0;
   PID[2].SP := 10.0;
   PID[3].SP := 0.0;
   PID[4].SP := 0.0;
   PID[5].SP := 0.0;
   PID[6].SP := 0.0;
   PID[7].SP := 0.0;
   PID[8].SP := 0.0;
   PID[9].SP := 0.0;
   PID[10].SP := 0.0;
   PID[11].SP := 0.0;
   PID[12].SP := 0.0;
   PID[13].SP := 0.0;
   PID[14].SP := 0.0;
   PID[15].SP := 0.0;
   PID[16].SP := 0.0;
   PID[17].SP := 0.0;
   PID[18].SP := 0.0;
   PID[19].SP := 0.0;
   PID[20].SP := 0.0;
   PID[21].SP := 0.0;
   PID[22].SP := 0.0;
   PID[23].SP := 0.0;
   PID[24].SP := 0.0;
   PID[25].SP := 0.0;
   PID[26].SP := 0.0;
   PID[27].SP := 0.0;
   PID[28].SP := 0.0;
   PID[29].SP := 0.0;
   PID[30].SP := 0.0;
   PID[31].SP := 0.0;
   PID[32].SP := 0.0;
   PID[33].SP := 0.0;
   PID[34].SP := 0.0;
   PID[35].SP := 0.0;
   PID[36].SP := 0.0;
   PID[37].SP := 0.0;
   PID[38].SP := 0.0;
   PID[39].SP := 0.0;
   PID[40].SP := 0.0;
   PID[41].SP := 0.0;
   PID[42].SP := 0.0;
   PID[43].SP := 0.0;
   PID[44].SP := 0.0;
   PID[45].SP := 0.0;
   PID[46].SP := 0.0;
   PID[47].SP := 0.0;
   PID[48].SP := 0.0;
   PID[49].SP := 0.0;
   PID[50].SP := 0.0;
   PID[51].SP := 0.0;
   PID[52].SP := 0.0;
   PID[53].SP := 0.0;
   PID[54].SP := 0.0;
   PID[55].SP := 70.0;
   PID[56].SP := 0.0;
   PID[57].SP := 0.0;
   PID[58].SP := 0.0;
   PID[59].SP := 0.0;
   PID[60].SP := 0.0;
   PID[61].SP := 0.0;
   PID[62].SP := 0.0;
   PID[63].SP := 0.0;
   PID[64].SP := 0.0;
   PID[65].SP := 0.0;
   PID[66].SP := 0.0;
   PID[67].SP := 0.0;
   PID[68].SP := 0.0;
   PID[69].SP := 0.0;
   PID[70].SP := 0.0;
   PID[71].SP := 0.0;
   PID[72].SP := 0.0;
   PID[73].SP := 0.0;
   PID[74].SP := 0.0;
   PID[75].SP := 0.0;
   PID[76].SP := 0.0;
   PID[77].SP := 0.0;
   PID[78].SP := 0.0;
   PID[79].SP := 0.0;
   PID[80].SP := 0.0;
   PID[81].SP := 0.0;
   PID[82].SP := 0.0;
   PID[83].SP := 0.0;
   PID[84].SP := 0.0;
   PID[85].SP := 0.0;
   PID[86].SP := 0.0;
   PID[87].SP := 0.0;
   PID[88].SP := 0.0;
   PID[89].SP := 0.0;
   PID[90].SP := 0.0;
   PID[91].SP := 0.0;
   PID[92].SP := 0.0;
   PID[93].SP := 0.0;
   PID[94].SP := 0.0;
   PID[95].SP := 0.0;
   PID[96].SP := 0.0;
   PID[97].SP := 0.0;
   PID[98].SP := 0.0;
   PID[99].SP := 0.0;
   PID[100].SP := 0.0;
END_DATA_BLOCK

DATA_BLOCK "ACESYS_HMI_PID_SPA_HLC"   // DB17
TITLE = ACESYS PID SPA-HLC DB
{ S7_Optimized_Access := 'FALSE' }
AUTHOR : METIS
FAMILY : ACESYS
NAME : PID_SP
VERSION : 8.0
   VAR
      PID : Array[0..100] of Struct   // Setpoint AUTO-HLC from HMI
         SP : Real;   // Auto HLC Setpoint Eng. Units
      END_STRUCT;
   END_VAR
BEGIN
   PID[0].SP := 0.0;
   PID[1].SP := 6.388889;
   PID[2].SP := 6.388888;
   PID[3].SP := 0.0;
   PID[4].SP := 7.398004;
   PID[5].SP := 7.398004;
   PID[6].SP := 0.07957175;
   PID[7].SP := 0.0;
   PID[8].SP := 0.0;
   PID[9].SP := 0.0;
   PID[10].SP := 0.0;
   PID[11].SP := 1.566117;
   PID[12].SP := 0.0;
   PID[13].SP := 1.388889;
   PID[14].SP := 0.0;
   PID[15].SP := 0.0;
   PID[16].SP := 0.0;
   PID[17].SP := 0.0;
   PID[18].SP := 0.0;
   PID[19].SP := 0.0;
   PID[20].SP := 0.0;
   PID[21].SP := 0.0;
   PID[22].SP := 0.0;
   PID[23].SP := 0.0;
   PID[24].SP := 0.0;
   PID[25].SP := 0.0;
   PID[26].SP := 0.0;
   PID[27].SP := 0.0;
   PID[28].SP := 0.0;
   PID[29].SP := 0.0;
   PID[30].SP := 0.0;
   PID[31].SP := 0.0;
   PID[32].SP := 0.0;
   PID[33].SP := 0.0;
   PID[34].SP := 0.0;
   PID[35].SP := 0.0;
   PID[36].SP := 0.0;
   PID[37].SP := 0.0;
   PID[38].SP := 0.0;
   PID[39].SP := 0.0;
   PID[40].SP := 0.0;
   PID[41].SP := 0.0;
   PID[42].SP := 0.0;
   PID[43].SP := 0.0;
   PID[44].SP := 0.0;
   PID[45].SP := 0.0;
   PID[46].SP := 0.0;
   PID[47].SP := 0.0;
   PID[48].SP := 0.0;
   PID[49].SP := 0.0;
   PID[50].SP := 0.0;
   PID[51].SP := 0.0;
   PID[52].SP := 0.0;
   PID[53].SP := 0.0;
   PID[54].SP := 0.0;
   PID[55].SP := 60.0;
   PID[56].SP := 0.0;
   PID[57].SP := 0.0;
   PID[58].SP := 0.0;
   PID[59].SP := 0.0;
   PID[60].SP := 0.0;
   PID[61].SP := 0.0;
   PID[62].SP := 0.0;
   PID[63].SP := 0.0;
   PID[64].SP := 0.0;
   PID[65].SP := 0.0;
   PID[66].SP := 0.0;
   PID[67].SP := 0.0;
   PID[68].SP := 0.0;
   PID[69].SP := 0.0;
   PID[70].SP := 0.0;
   PID[71].SP := 0.0;
   PID[72].SP := 0.0;
   PID[73].SP := 0.0;
   PID[74].SP := 0.0;
   PID[75].SP := 0.0;
   PID[76].SP := 0.0;
   PID[77].SP := 0.0;
   PID[78].SP := 0.0;
   PID[79].SP := 0.0;
   PID[80].SP := 0.0;
   PID[81].SP := 0.0;
   PID[82].SP := 0.0;
   PID[83].SP := 0.0;
   PID[84].SP := 0.0;
   PID[85].SP := 0.0;
   PID[86].SP := 0.0;
   PID[87].SP := 0.0;
   PID[88].SP := 0.0;
   PID[89].SP := 0.0;
   PID[90].SP := 0.0;
   PID[91].SP := 0.0;
   PID[92].SP := 0.0;
   PID[93].SP := 0.0;
   PID[94].SP := 0.0;
   PID[95].SP := 0.0;
   PID[96].SP := 0.0;
   PID[97].SP := 0.0;
   PID[98].SP := 0.0;
   PID[99].SP := 0.0;
   PID[100].SP := 0.0;
END_DATA_BLOCK

DATA_BLOCK "ACESYS_HMI_PID_SPM_HLC"   // DB18
TITLE = ACESYS PID SPM-HLC DB
{ S7_Optimized_Access := 'FALSE' }
AUTHOR : METIS
FAMILY : ACESYS
NAME : PID_SP
VERSION : 8.0
   VAR
      PID : Array[0..100] of Struct   // Setpoint MAN-HLC from HMI
         SP : Real;   // MANUAL HLC Setpoint in Pct
      END_STRUCT;
   END_VAR
BEGIN
   PID[0].SP := 0.0;
   PID[1].SP := 100.0;
   PID[2].SP := 10.0;
   PID[3].SP := 0.0;
   PID[4].SP := 0.0;
   PID[5].SP := 0.0;
   PID[6].SP := 0.0;
   PID[7].SP := 0.0;
   PID[8].SP := 0.0;
   PID[9].SP := 0.0;
   PID[10].SP := 0.0;
   PID[11].SP := 0.0;
   PID[12].SP := 0.0;
   PID[13].SP := 0.0;
   PID[14].SP := 0.0;
   PID[15].SP := 0.0;
   PID[16].SP := 0.0;
   PID[17].SP := 0.0;
   PID[18].SP := 0.0;
   PID[19].SP := 0.0;
   PID[20].SP := 0.0;
   PID[21].SP := 0.0;
   PID[22].SP := 0.0;
   PID[23].SP := 0.0;
   PID[24].SP := 0.0;
   PID[25].SP := 0.0;
   PID[26].SP := 0.0;
   PID[27].SP := 0.0;
   PID[28].SP := 0.0;
   PID[29].SP := 0.0;
   PID[30].SP := 0.0;
   PID[31].SP := 0.0;
   PID[32].SP := 0.0;
   PID[33].SP := 0.0;
   PID[34].SP := 0.0;
   PID[35].SP := 0.0;
   PID[36].SP := 0.0;
   PID[37].SP := 0.0;
   PID[38].SP := 0.0;
   PID[39].SP := 0.0;
   PID[40].SP := 0.0;
   PID[41].SP := 0.0;
   PID[42].SP := 0.0;
   PID[43].SP := 0.0;
   PID[44].SP := 0.0;
   PID[45].SP := 0.0;
   PID[46].SP := 0.0;
   PID[47].SP := 0.0;
   PID[48].SP := 0.0;
   PID[49].SP := 0.0;
   PID[50].SP := 0.0;
   PID[51].SP := 0.0;
   PID[52].SP := 0.0;
   PID[53].SP := 0.0;
   PID[54].SP := 0.0;
   PID[55].SP := 70.0;
   PID[56].SP := 0.0;
   PID[57].SP := 0.0;
   PID[58].SP := 0.0;
   PID[59].SP := 0.0;
   PID[60].SP := 0.0;
   PID[61].SP := 0.0;
   PID[62].SP := 0.0;
   PID[63].SP := 0.0;
   PID[64].SP := 0.0;
   PID[65].SP := 0.0;
   PID[66].SP := 0.0;
   PID[67].SP := 0.0;
   PID[68].SP := 0.0;
   PID[69].SP := 0.0;
   PID[70].SP := 0.0;
   PID[71].SP := 0.0;
   PID[72].SP := 0.0;
   PID[73].SP := 0.0;
   PID[74].SP := 0.0;
   PID[75].SP := 0.0;
   PID[76].SP := 0.0;
   PID[77].SP := 0.0;
   PID[78].SP := 0.0;
   PID[79].SP := 0.0;
   PID[80].SP := 0.0;
   PID[81].SP := 0.0;
   PID[82].SP := 0.0;
   PID[83].SP := 0.0;
   PID[84].SP := 0.0;
   PID[85].SP := 0.0;
   PID[86].SP := 0.0;
   PID[87].SP := 0.0;
   PID[88].SP := 0.0;
   PID[89].SP := 0.0;
   PID[90].SP := 0.0;
   PID[91].SP := 0.0;
   PID[92].SP := 0.0;
   PID[93].SP := 0.0;
   PID[94].SP := 0.0;
   PID[95].SP := 0.0;
   PID[96].SP := 0.0;
   PID[97].SP := 0.0;
   PID[98].SP := 0.0;
   PID[99].SP := 0.0;
   PID[100].SP := 0.0;
END_DATA_BLOCK

DATA_BLOCK "CNT_Storage_DB"   // DB71
{ S7_Optimized_Access := 'FALSE' }
VERSION : 0.1
   VAR
      Data : Array[0..70] of "CNT_for_Period";
   END_VAR
BEGIN
   Data[0].CNT_Begin := 0.0;
   Data[0].CNT_Current := 0.0;   // 2090PU735N01F01_Cnt_CurDay
   Data[0].CNT_Previous := 0.0;   // 2090PU735N01F01_PrevDay
   Data[1].CNT_Begin := 0.0;
   Data[1].CNT_Current := 0.0;
   Data[1].CNT_Previous := 0.0;
   Data[2].CNT_Begin := 0.0;
   Data[2].CNT_Current := 0.0;
   Data[2].CNT_Previous := 0.0;
   Data[3].CNT_Begin := 0.0;
   Data[3].CNT_Current := 0.0;
   Data[3].CNT_Previous := 0.0;
   Data[4].CNT_Begin := 0.0;
   Data[4].CNT_Current := 0.0;
   Data[4].CNT_Previous := 0.0;
   Data[5].CNT_Begin := 0.0;
   Data[5].CNT_Current := 0.0;
   Data[5].CNT_Previous := 0.0;
   Data[6].CNT_Begin := 0.0;
   Data[6].CNT_Current := 0.0;
   Data[6].CNT_Previous := 0.0;
   Data[7].CNT_Begin := 0.0;
   Data[7].CNT_Current := 0.0;
   Data[7].CNT_Previous := 0.0;
   Data[8].CNT_Begin := 0.0;
   Data[8].CNT_Current := 0.0;
   Data[8].CNT_Previous := 0.0;
   Data[9].CNT_Begin := 0.0;
   Data[9].CNT_Current := 0.0;
   Data[9].CNT_Previous := 0.0;
   Data[10].CNT_Begin := 0.0;
   Data[10].CNT_Current := 0.0;
   Data[10].CNT_Previous := 0.0;
   Data[11].CNT_Begin := 0.0;
   Data[11].CNT_Current := 0.0;
   Data[11].CNT_Previous := 0.0;
   Data[12].CNT_Begin := 0.0;
   Data[12].CNT_Current := 0.0;
   Data[12].CNT_Previous := 0.0;
   Data[13].CNT_Begin := 0.0;
   Data[13].CNT_Current := 0.0;
   Data[13].CNT_Previous := 0.0;
   Data[14].CNT_Begin := 0.0;
   Data[14].CNT_Current := 0.0;
   Data[14].CNT_Previous := 0.0;
   Data[15].CNT_Begin := 0.0;
   Data[15].CNT_Current := 0.0;
   Data[15].CNT_Previous := 0.0;
   Data[16].CNT_Begin := 0.0;
   Data[16].CNT_Current := 0.0;
   Data[16].CNT_Previous := 0.0;
   Data[17].CNT_Begin := 0.0;
   Data[17].CNT_Current := 0.0;
   Data[17].CNT_Previous := 0.0;
   Data[18].CNT_Begin := 0.0;
   Data[18].CNT_Current := 0.0;
   Data[18].CNT_Previous := 0.0;
   Data[19].CNT_Begin := 0.0;
   Data[19].CNT_Current := 0.0;
   Data[19].CNT_Previous := 0.0;
   Data[20].CNT_Begin := 0.0;
   Data[20].CNT_Current := 0.0;
   Data[20].CNT_Previous := 0.0;
   Data[21].CNT_Begin := 0.0;
   Data[21].CNT_Current := 0.0;
   Data[21].CNT_Previous := 0.0;
   Data[22].CNT_Begin := 0.0;
   Data[22].CNT_Current := 0.0;
   Data[22].CNT_Previous := 0.0;
   Data[23].CNT_Begin := 0.0;
   Data[23].CNT_Current := 0.0;
   Data[23].CNT_Previous := 0.0;
   Data[24].CNT_Begin := 0.0;
   Data[24].CNT_Current := 0.0;
   Data[24].CNT_Previous := 0.0;
   Data[25].CNT_Begin := 0.0;
   Data[25].CNT_Current := 0.0;
   Data[25].CNT_Previous := 0.0;
   Data[26].CNT_Begin := 0.0;
   Data[26].CNT_Current := 0.0;
   Data[26].CNT_Previous := 0.0;
   Data[27].CNT_Begin := 0.0;
   Data[27].CNT_Current := 0.0;
   Data[27].CNT_Previous := 0.0;
   Data[28].CNT_Begin := 0.0;
   Data[28].CNT_Current := 0.0;
   Data[28].CNT_Previous := 0.0;
   Data[29].CNT_Begin := 0.0;
   Data[29].CNT_Current := 0.0;
   Data[29].CNT_Previous := 0.0;
   Data[30].CNT_Begin := 0.0;
   Data[30].CNT_Current := 0.0;
   Data[30].CNT_Previous := 0.0;
   Data[31].CNT_Begin := 0.0;
   Data[31].CNT_Current := 0.0;
   Data[31].CNT_Previous := 0.0;
   Data[32].CNT_Begin := 0.0;
   Data[32].CNT_Current := 0.0;
   Data[32].CNT_Previous := 0.0;
   Data[33].CNT_Begin := 0.0;
   Data[33].CNT_Current := 0.0;
   Data[33].CNT_Previous := 0.0;
   Data[34].CNT_Begin := 0.0;
   Data[34].CNT_Current := 0.0;
   Data[34].CNT_Previous := 0.0;
   Data[35].CNT_Begin := 0.0;
   Data[35].CNT_Current := 0.0;
   Data[35].CNT_Previous := 0.0;
   Data[36].CNT_Begin := 0.0;
   Data[36].CNT_Current := 0.0;
   Data[36].CNT_Previous := 0.0;
   Data[37].CNT_Begin := 0.0;
   Data[37].CNT_Current := 0.0;
   Data[37].CNT_Previous := 0.0;
   Data[38].CNT_Begin := 0.0;
   Data[38].CNT_Current := 0.0;
   Data[38].CNT_Previous := 0.0;
   Data[39].CNT_Begin := 0.0;
   Data[39].CNT_Current := 0.0;
   Data[39].CNT_Previous := 0.0;
   Data[40].CNT_Begin := 0.0;
   Data[40].CNT_Current := 0.0;
   Data[40].CNT_Previous := 0.0;
   Data[41].CNT_Begin := 0.0;
   Data[41].CNT_Current := 0.0;
   Data[41].CNT_Previous := 0.0;
   Data[42].CNT_Begin := 0.0;
   Data[42].CNT_Current := 0.0;
   Data[42].CNT_Previous := 0.0;
   Data[43].CNT_Begin := 0.0;
   Data[43].CNT_Current := 0.0;
   Data[43].CNT_Previous := 0.0;
   Data[44].CNT_Begin := 0.0;
   Data[44].CNT_Current := 0.0;
   Data[44].CNT_Previous := 0.0;
   Data[45].CNT_Begin := 0.0;
   Data[45].CNT_Current := 0.0;
   Data[45].CNT_Previous := 0.0;
   Data[46].CNT_Begin := 0.0;
   Data[46].CNT_Current := 0.0;
   Data[46].CNT_Previous := 0.0;
   Data[47].CNT_Begin := 0.0;
   Data[47].CNT_Current := 0.0;
   Data[47].CNT_Previous := 0.0;
   Data[48].CNT_Begin := 0.0;
   Data[48].CNT_Current := 0.0;
   Data[48].CNT_Previous := 0.0;
   Data[49].CNT_Begin := 0.0;
   Data[49].CNT_Current := 0.0;
   Data[49].CNT_Previous := 0.0;
   Data[50].CNT_Begin := 0.0;
   Data[50].CNT_Current := 0.0;
   Data[50].CNT_Previous := 0.0;
   Data[51].CNT_Begin := 0.0;
   Data[51].CNT_Current := 0.0;
   Data[51].CNT_Previous := 0.0;
   Data[52].CNT_Begin := 0.0;
   Data[52].CNT_Current := 0.0;
   Data[52].CNT_Previous := 0.0;
   Data[53].CNT_Begin := 0.0;
   Data[53].CNT_Current := 0.0;
   Data[53].CNT_Previous := 0.0;
   Data[54].CNT_Begin := 0.0;
   Data[54].CNT_Current := 0.0;
   Data[54].CNT_Previous := 0.0;
   Data[55].CNT_Begin := 0.0;
   Data[55].CNT_Current := 0.0;
   Data[55].CNT_Previous := 0.0;
   Data[56].CNT_Begin := 0.0;
   Data[56].CNT_Current := 0.0;
   Data[56].CNT_Previous := 0.0;
   Data[57].CNT_Begin := 0.0;
   Data[57].CNT_Current := 0.0;
   Data[57].CNT_Previous := 0.0;
   Data[58].CNT_Begin := 0.0;
   Data[58].CNT_Current := 0.0;
   Data[58].CNT_Previous := 0.0;
   Data[59].CNT_Begin := 0.0;
   Data[59].CNT_Current := 0.0;
   Data[59].CNT_Previous := 0.0;
   Data[60].CNT_Begin := 0.0;
   Data[60].CNT_Current := 0.0;
   Data[60].CNT_Previous := 0.0;
   Data[61].CNT_Begin := 0.0;
   Data[61].CNT_Current := 0.0;
   Data[61].CNT_Previous := 0.0;
   Data[62].CNT_Begin := 0.0;
   Data[62].CNT_Current := 0.0;
   Data[62].CNT_Previous := 0.0;
   Data[63].CNT_Begin := 0.0;
   Data[63].CNT_Current := 0.0;
   Data[63].CNT_Previous := 0.0;
   Data[64].CNT_Begin := 0.0;
   Data[64].CNT_Current := 0.0;
   Data[64].CNT_Previous := 0.0;
   Data[65].CNT_Begin := 0.0;
   Data[65].CNT_Current := 0.0;
   Data[65].CNT_Previous := 0.0;
   Data[66].CNT_Begin := 0.0;
   Data[66].CNT_Current := 0.0;
   Data[66].CNT_Previous := 0.0;
   Data[67].CNT_Begin := 0.0;
   Data[67].CNT_Current := 0.0;
   Data[67].CNT_Previous := 0.0;
   Data[68].CNT_Begin := 0.0;
   Data[68].CNT_Current := 0.0;
   Data[68].CNT_Previous := 0.0;
   Data[69].CNT_Begin := 0.0;
   Data[69].CNT_Current := 0.0;
   Data[69].CNT_Previous := 0.0;
   Data[70].CNT_Begin := 0.0;
   Data[70].CNT_Current := 0.0;
   Data[70].CNT_Previous := 0.0;
   // Data[0] : 2090PU735N01F01_TOT
END_DATA_BLOCK

